C09100=1017.459,-55.888,398.347,165.702,54.848,159.813
C09101=1017.465,-55.638,398.336,165.706,54.842,159.813
C09102=1017.470,-55.388,398.326,165.708,54.836,159.812
C09103=1017.475,-55.139,398.315,165.712,54.830,159.812
C09104=1017.481,-54.889,398.305,165.714,54.824,159.811
C09105=1017.486,-54.640,398.294,165.717,54.817,159.810
C09106=1017.491,-54.389,398.284,165.721,54.811,159.810
C09107=1017.497,-54.140,398.273,165.723,54.805,159.810
C09108=1017.503,-53.863,398.261,165.726,54.798,159.809
C09109=1017.509,-53.585,398.250,165.729,54.791,159.808
C09110=1017.515,-53.308,398.237,165.733,54.784,159.808
C09111=1017.522,-53.030,398.226,165.737,54.777,159.808
C09112=1017.527,-52.780,398.216,165.739,54.771,159.807
C09113=1017.533,-52.531,398.205,165.741,54.765,159.806
C09114=1017.539,-52.281,398.194,165.745,54.759,159.806
C09115=1017.543,-52.032,398.184,165.748,54.752,159.805
C09116=1017.549,-51.782,398.173,165.751,54.746,159.805
C09117=1017.554,-51.532,398.162,165.753,54.739,159.804
C09118=1017.560,-51.282,398.151,165.757,54.733,159.804
C09119=1017.565,-51.033,398.141,165.759,54.727,159.803
C09120=1017.571,-50.783,398.130,165.762,54.721,159.803
C09121=1017.576,-50.533,398.118,165.766,54.715,159.803
C09122=1017.582,-50.283,398.108,165.768,54.709,159.802
C09123=1017.587,-50.034,398.097,165.771,54.703,159.802
C09124=1017.592,-49.784,398.086,165.775,54.697,159.801
C09125=1017.597,-49.534,398.074,165.777,54.691,159.801
C09126=1017.603,-49.285,398.063,165.780,54.685,159.800
C09127=1017.608,-49.035,398.052,165.783,54.678,159.800
C09128=1017.614,-48.785,398.041,165.786,54.673,159.799
C09129=1017.619,-48.536,398.030,165.789,54.667,159.799
C09130=1017.625,-48.286,398.019,165.791,54.661,159.798
C09131=1017.630,-48.036,398.007,165.795,54.655,159.798
C09132=1017.635,-47.787,397.996,165.797,54.649,159.797
C09133=1017.640,-47.536,397.986,165.800,54.643,159.797
C09134=1017.646,-47.287,397.975,165.803,54.636,159.797
C09135=1017.651,-47.037,397.963,165.806,54.631,159.796
C09136=1017.656,-46.788,397.952,165.808,54.624,159.796
C09137=1017.661,-46.538,397.941,165.812,54.618,159.795
C09138=1017.667,-46.288,397.930,165.815,54.612,159.795
C09139=1017.672,-46.039,397.919,165.817,54.606,159.794
C09140=1017.678,-45.789,397.908,165.821,54.600,159.794
C09141=1017.683,-45.539,397.896,165.823,54.594,159.793
C09142=1017.689,-45.289,397.885,165.826,54.588,159.793
C09143=1017.694,-45.039,397.873,165.828,54.582,159.792
C09144=1017.700,-44.790,397.863,165.832,54.576,159.792
C09145=1017.705,-44.540,397.851,165.834,54.570,159.791
C09146=1017.711,-44.291,397.840,165.837,54.563,159.791
C09147=1017.716,-44.041,397.829,165.841,54.557,159.790
C09148=1017.722,-43.792,397.817,165.843,54.551,159.790
C09149=1017.727,-43.542,397.806,165.846,54.546,159.789
C09150=1017.733,-43.293,397.795,165.849,54.539,159.789
C09151=1017.738,-43.043,397.783,165.852,54.533,159.789
C09152=1017.744,-42.793,397.772,165.854,54.527,159.788
C09153=1017.749,-42.543,397.761,165.858,54.520,159.787
C09154=1017.755,-42.293,397.750,165.861,54.515,159.787
C09155=1017.760,-42.043,397.738,165.864,54.508,159.787
C09156=1017.765,-41.794,397.727,165.866,54.502,159.786
C09157=1017.770,-41.544,397.716,165.869,54.496,159.785
C09158=1017.776,-41.295,397.705,165.873,54.490,159.785
C09159=1017.782,-41.045,397.693,165.875,54.483,159.784
C09160=1017.788,-40.795,397.682,165.878,54.478,159.784
C09161=1017.793,-40.546,397.670,165.881,54.471,159.783
C09162=1017.798,-40.296,397.659,165.883,54.465,159.783
C09163=1017.803,-40.046,397.648,165.886,54.459,159.782
C09164=1017.809,-39.797,397.637,165.890,54.453,159.782
C09165=1017.815,-39.547,397.624,165.892,54.446,159.781
C09166=1017.820,-39.297,397.613,165.895,54.441,159.781
C09167=1017.826,-39.048,397.602,165.898,54.434,159.780
C09168=1017.831,-38.798,397.591,165.901,54.429,159.780
C09169=1017.836,-38.549,397.578,165.903,54.422,159.779
C09170=1017.842,-38.298,397.567,165.906,54.417,159.779
C09171=1017.847,-38.048,397.555,165.910,54.410,159.779
C09172=1017.853,-37.772,397.542,165.913,54.404,159.778
C09173=1017.859,-37.495,397.529,165.915,54.397,159.777
C09174=1017.865,-37.217,397.516,165.919,54.391,159.777
C09175=1017.871,-36.940,397.503,165.922,54.384,159.776
C09176=1017.876,-36.690,397.491,165.924,54.378,159.776
C09177=1017.882,-36.441,397.480,165.928,54.371,159.775
C09178=1017.887,-36.191,397.468,165.931,54.366,159.775
C09179=1017.893,-35.942,397.456,165.933,54.359,159.774
C09180=1017.898,-35.691,397.444,165.936,54.354,159.774
C09181=1017.904,-35.442,397.434,165.939,54.347,159.773
C09182=1017.909,-35.193,397.421,165.942,54.342,159.773
C09183=1017.914,-34.943,397.410,165.945,54.335,159.772
C09184=1017.920,-34.693,397.397,165.948,54.329,159.772
C09185=1017.925,-34.443,397.386,165.951,54.323,159.771
C09186=1017.931,-34.194,397.374,165.953,54.317,159.771
C09187=1017.937,-33.944,397.362,165.955,54.311,159.770
C09188=1017.942,-33.695,397.350,165.959,54.305,159.770
C09189=1017.947,-33.445,397.339,165.962,54.298,159.769
C09190=1017.952,-33.196,397.327,165.965,54.293,159.769
C09191=1017.959,-32.945,397.315,165.968,54.286,159.768
C09192=1017.964,-32.696,397.303,165.970,54.280,159.768
C09193=1017.969,-32.446,397.292,165.973,54.274,159.767
C09194=1017.975,-32.197,397.279,165.976,54.268,159.767
C09195=1017.980,-31.947,397.268,165.979,54.262,159.766
C09196=1017.985,-31.698,397.255,165.982,54.256,159.766
C09197=1017.992,-31.447,397.244,165.984,54.250,159.765
C09198=1017.997,-31.198,397.232,165.988,54.243,159.765
C09199=1018.002,-30.948,397.221,165.990,54.238,159.764
C09200=1018.008,-30.698,397.208,165.993,54.231,159.764
C09201=1018.013,-30.449,397.197,165.996,54.225,159.763
C09202=1018.020,-30.199,397.185,165.999,54.219,159.763
C09203=1018.025,-29.949,397.173,166.001,54.213,159.762
C09204=1018.030,-29.700,397.161,166.004,54.207,159.761
C09205=1018.036,-29.450,397.148,166.007,54.200,159.761
C09206=1018.041,-29.200,397.137,166.010,54.195,159.761
C09207=1018.047,-28.951,397.125,166.012,54.188,159.760
C09208=1018.052,-28.701,397.113,166.016,54.182,159.759
C09209=1018.058,-28.452,397.101,166.018,54.176,159.759
C09210=1018.064,-28.202,397.089,166.021,54.169,159.758
C09211=1018.069,-27.952,397.077,166.025,54.163,159.758
C09212=1018.075,-27.702,397.065,166.027,54.157,159.757
C09213=1018.080,-27.452,397.053,166.029,54.151,159.757
C09214=1018.085,-27.203,397.041,166.032,54.145,159.756
C09215=1018.091,-26.953,397.028,166.036,54.139,159.756
C09216=1018.096,-26.704,397.016,166.038,54.133,159.755
C09217=1018.102,-26.454,397.004,166.041,54.127,159.755
C09218=1018.107,-26.205,396.992,166.043,54.121,159.754
C09219=1018.113,-25.955,396.980,166.047,54.115,159.754
C09220=1018.118,-25.706,396.968,166.050,54.109,159.753
C09221=1018.124,-25.456,396.955,166.052,54.103,159.753
C09222=1018.129,-25.206,396.943,166.055,54.097,159.752
C09223=1018.134,-24.956,396.930,166.057,54.091,159.751
C09224=1018.140,-24.706,396.918,166.061,54.085,159.751
C09225=1018.145,-24.457,396.906,166.063,54.079,159.751
C09226=1018.151,-24.207,396.893,166.066,54.072,159.750
C09227=1018.156,-23.958,396.881,166.069,54.067,159.750
C09228=1018.162,-23.708,396.869,166.072,54.060,159.749
C09229=1018.167,-23.459,396.856,166.075,54.055,159.749
C09230=1018.173,-23.209,396.845,166.077,54.049,159.748
C09231=1018.178,-22.959,396.832,166.080,54.042,159.747
C09232=1018.184,-22.710,396.820,166.083,54.036,159.747
C09233=1018.189,-22.460,396.807,166.086,54.030,159.746
C09234=1018.195,-22.210,396.795,166.089,54.024,159.746
C09235=1018.200,-21.961,396.782,166.091,54.018,159.745
C09236=1018.206,-21.683,396.769,166.094,54.011,159.745
C09237=1018.213,-21.405,396.754,166.098,54.005,159.744
C09238=1018.219,-21.127,396.741,166.101,53.997,159.743
C09239=1018.225,-20.848,396.727,166.104,53.991,159.743
C09240=1018.230,-20.598,396.714,166.107,53.984,159.742
C09241=1018.236,-20.349,396.702,166.109,53.978,159.742
C09242=1018.242,-20.099,396.690,166.112,53.973,159.741
C09243=1018.247,-19.850,396.678,166.115,53.966,159.741
C09244=1018.253,-19.600,396.665,166.118,53.960,159.740
C09245=1018.258,-19.351,396.653,166.120,53.954,159.740
C09246=1018.264,-19.101,396.640,166.123,53.948,159.739
C09247=1018.269,-18.851,396.627,166.126,53.942,159.739
C09248=1018.275,-18.602,396.615,166.129,53.935,159.738
C09249=1018.280,-18.352,396.602,166.131,53.929,159.737
C09250=1018.286,-18.103,396.590,166.134,53.924,159.737
C09251=1018.292,-17.853,396.578,166.138,53.917,159.736
C09252=1018.298,-17.603,396.565,166.140,53.911,159.736
C09253=1018.303,-17.354,396.553,166.142,53.905,159.735
C09254=1018.309,-17.104,396.540,166.146,53.898,159.735
C09255=1018.314,-16.855,396.528,166.149,53.893,159.734
C09256=1018.319,-16.605,396.515,166.151,53.886,159.734
C09257=1018.325,-16.355,396.502,166.154,53.880,159.733
C09258=1018.331,-16.106,396.490,166.157,53.874,159.732
C09259=1018.336,-15.856,396.478,166.159,53.867,159.732
C09260=1018.343,-15.606,396.464,166.162,53.862,159.731
C09261=1018.347,-15.357,396.452,166.165,53.856,159.731
C09262=1018.353,-15.107,396.439,166.167,53.850,159.730
C09263=1018.358,-14.857,396.426,166.171,53.844,159.730
C09264=1018.364,-14.608,396.413,166.174,53.837,159.729
C09265=1018.370,-14.358,396.400,166.176,53.831,159.729
C09266=1018.374,-14.109,396.388,166.179,53.826,159.728
C09267=1018.380,-13.859,396.375,166.181,53.820,159.728
C09268=1018.388,-13.518,396.357,166.185,53.811,159.727
C09269=1018.396,-13.177,396.340,166.188,53.803,159.726
C09270=1018.403,-12.835,396.322,166.194,53.795,159.725
C09271=1018.410,-12.493,396.304,166.197,53.786,159.725
C09272=1018.416,-12.245,396.291,166.200,53.780,159.724
C09273=1018.421,-11.995,396.278,166.202,53.774,159.723
C09274=1018.427,-11.745,396.266,166.205,53.769,159.723
C09275=1018.433,-11.496,396.253,166.207,53.762,159.722
C09276=1018.438,-11.246,396.240,166.211,53.756,159.722
C09277=1018.444,-10.996,396.227,166.213,53.750,159.721
C09278=1018.449,-10.747,396.214,166.216,53.743,159.721
C09279=1018.455,-10.497,396.201,166.218,53.738,159.720
C09280=1018.460,-10.247,396.189,166.221,53.732,159.719
C09281=1018.466,-9.998,396.175,166.224,53.725,159.719
C09282=1018.471,-9.749,396.163,166.227,53.719,159.718
C09283=1018.476,-9.499,396.149,166.230,53.714,159.718
C09284=1018.483,-9.249,396.136,166.232,53.707,159.717
C09285=1018.489,-8.999,396.124,166.235,53.701,159.717
C09286=1018.493,-8.751,396.110,166.238,53.695,159.716
C09287=1018.499,-8.501,396.097,166.241,53.688,159.716
C09288=1018.505,-8.250,396.084,166.243,53.683,159.715
C09289=1018.511,-8.001,396.071,166.246,53.677,159.714
C09290=1018.517,-7.751,396.059,166.248,53.671,159.714
C09291=1018.522,-7.502,396.045,166.252,53.664,159.713
C09292=1018.527,-7.253,396.032,166.254,53.658,159.713
C09293=1018.533,-7.003,396.019,166.257,53.652,159.712
C09294=1018.539,-6.753,396.006,166.259,53.646,159.711
C09295=1018.544,-6.503,395.993,166.263,53.640,159.711
C09296=1018.549,-6.285,395.982,166.264,53.634,159.710
C09297=1018.554,-6.066,395.970,166.267,53.628,159.710
C09298=1018.559,-5.847,395.959,166.269,53.623,159.709
C09299=1018.563,-5.628,395.947,166.272,53.618,159.709
C09300=1018.569,-5.409,395.936,166.275,53.612,159.709
C09301=1018.574,-5.191,395.924,166.277,53.607,159.708
C09302=1018.578,-4.971,395.913,166.279,53.601,159.707
C09303=1018.583,-4.752,395.902,166.281,53.596,159.707
C09304=1018.590,-4.503,395.888,166.285,53.590,159.706
C09305=1018.595,-4.253,395.875,166.287,53.583,159.706
C09306=1018.600,-4.003,395.861,166.290,53.578,159.705
C09307=1018.606,-3.754,395.848,166.293,53.572,159.705
C09308=1018.612,-3.504,395.835,166.295,53.566,159.704
C09309=1018.617,-3.254,395.821,166.298,53.560,159.703
C09310=1018.622,-3.005,395.807,166.300,53.554,159.703
C09311=1018.628,-2.755,395.795,166.303,53.548,159.702
C09312=1018.633,-2.506,395.781,166.306,53.542,159.702
C09313=1018.639,-2.256,395.767,166.308,53.536,159.701
C09314=1018.644,-2.007,395.753,166.312,53.530,159.701
C09315=1018.649,-1.757,395.740,166.315,53.524,159.700
C09316=1018.656,-1.507,395.727,166.317,53.518,159.700
C09317=1018.660,-1.258,395.713,166.319,53.512,159.699
C09318=1018.666,-1.009,395.700,166.322,53.506,159.698
C09319=1018.671,-0.759,395.686,166.325,53.500,159.698
C09320=1018.677,-0.509,395.673,166.327,53.494,159.697
C09321=1018.683,-0.260,395.659,166.330,53.488,159.697
C09322=1018.688,-0.010,395.645,166.333,53.483,159.696
C09323=1018.694,0.239,395.632,166.336,53.476,159.696
C09324=1018.699,0.490,395.618,166.339,53.470,159.695
C09325=1018.705,0.739,395.605,166.341,53.464,159.694
C09326=1018.711,0.988,395.591,166.344,53.458,159.694
C09327=1018.716,1.238,395.577,166.347,53.452,159.693
C09328=1018.721,1.487,395.564,166.349,53.446,159.693
C09329=1018.726,1.737,395.551,166.351,53.440,159.692
C09330=1018.732,1.986,395.537,166.354,53.434,159.691
C09331=1018.738,2.236,395.524,166.358,53.428,159.691
C09332=1018.743,2.485,395.510,166.360,53.422,159.690
C09333=1018.749,2.735,395.496,166.363,53.416,159.690
C09334=1018.754,2.985,395.482,166.365,53.409,159.689
C09335=1018.760,3.234,395.469,166.368,53.403,159.688
C09336=1018.766,3.484,395.456,166.370,53.397,159.688
C09337=1018.771,3.734,395.442,166.373,53.392,159.687
C09338=1018.777,3.983,395.428,166.376,53.386,159.687
C09339=1018.782,4.233,395.414,166.379,53.379,159.686
C09340=1018.788,4.482,395.401,166.382,53.373,159.686
C09341=1018.794,4.732,395.387,166.384,53.367,159.685
C09342=1018.799,4.981,395.373,166.387,53.361,159.684
C09343=1018.805,5.231,395.359,166.389,53.354,159.684
C09344=1018.810,5.480,395.345,166.392,53.348,159.683
C09345=1018.816,5.730,395.332,166.395,53.343,159.683
C09346=1018.822,5.980,395.319,166.398,53.336,159.682
C09347=1018.827,6.229,395.305,166.401,53.330,159.681
C09348=1018.833,6.479,395.291,166.403,53.324,159.681
C09349=1018.838,6.729,395.277,166.405,53.318,159.680
C09350=1018.844,6.978,395.264,166.408,53.312,159.680
C09351=1018.850,7.227,395.250,166.410,53.306,159.679
C09352=1018.855,7.477,395.236,166.414,53.299,159.678
C09353=1018.861,7.727,395.222,166.416,53.293,159.678
C09354=1018.866,7.976,395.209,166.419,53.287,159.677
C09355=1018.872,8.225,395.195,166.421,53.281,159.676
C09356=1018.878,8.475,395.181,166.424,53.275,159.676
C09357=1018.883,8.724,395.168,166.426,53.269,159.675
C09358=1018.889,8.975,395.153,166.430,53.262,159.675
C09359=1018.895,9.224,395.139,166.433,53.257,159.674
C09360=1018.901,9.474,395.126,166.435,53.250,159.674
C09361=1018.907,9.723,395.112,166.438,53.244,159.673
C09362=1018.912,9.973,395.098,166.440,53.238,159.672
C09363=1018.917,10.222,395.085,166.443,53.232,159.672
C09364=1018.924,10.503,395.069,166.446,53.225,159.671
C09365=1018.930,10.785,395.053,166.449,53.218,159.670
C09366=1018.937,11.067,395.038,166.452,53.210,159.669
C09367=1018.944,11.349,395.022,166.455,53.203,159.669
C09368=1018.949,11.599,395.008,166.458,53.197,159.668
C09369=1018.955,11.849,394.994,166.460,53.191,159.667
C09370=1018.961,12.098,394.981,166.463,53.185,159.667
C09371=1018.966,12.347,394.967,166.466,53.178,159.666
C09372=1018.972,12.597,394.953,166.469,53.172,159.666
C09373=1018.977,12.847,394.939,166.471,53.166,159.665
C09374=1018.983,13.096,394.925,166.474,53.160,159.664
C09375=1018.989,13.346,394.910,166.476,53.154,159.664
C09376=1018.995,13.595,394.896,166.479,53.148,159.663
C09377=1019.000,13.845,394.882,166.482,53.141,159.663
C09378=1019.006,14.094,394.869,166.485,53.135,159.662
C09379=1019.011,14.343,394.854,166.488,53.130,159.661
C09380=1019.017,14.593,394.840,166.490,53.124,159.661
C09381=1019.022,14.843,394.826,166.493,53.118,159.660
C09382=1019.029,15.092,394.811,166.495,53.111,159.659
C09383=1019.034,15.342,394.797,166.498,53.105,159.659
C09384=1019.039,15.592,394.783,166.500,53.099,159.658
C09385=1019.044,15.841,394.769,166.503,53.093,159.658
C09386=1019.050,16.090,394.755,166.505,53.087,159.657
C09387=1019.056,16.340,394.741,166.509,53.081,159.656
C09388=1019.062,16.590,394.726,166.511,53.074,159.656
C09389=1019.067,16.839,394.712,166.514,53.068,159.655
C09390=1019.073,17.089,394.698,166.516,53.062,159.654
C09391=1019.079,17.338,394.683,166.519,53.056,159.654
C09392=1019.084,17.587,394.670,166.521,53.050,159.653
C09393=1019.090,17.838,394.655,166.524,53.045,159.653
C09394=1019.095,18.087,394.640,166.527,53.039,159.652
C09395=1019.101,18.336,394.626,166.529,53.032,159.651
C09396=1019.106,18.586,394.612,166.533,53.026,159.651
C09397=1019.113,18.835,394.597,166.536,53.020,159.650
C09398=1019.118,19.085,394.584,166.538,53.014,159.650
C09399=1019.124,19.334,394.569,166.541,53.008,159.649
C09400=1019.129,19.584,394.555,166.543,53.002,159.648
C09401=1019.134,19.833,394.540,166.546,52.995,159.648
C09402=1019.141,20.083,394.526,166.548,52.989,159.647
C09403=1019.146,20.332,394.511,166.551,52.983,159.646
C09404=1019.151,20.582,394.497,166.553,52.977,159.646
C09405=1019.157,20.831,394.482,166.556,52.971,159.645
C09406=1019.163,21.081,394.468,166.558,52.965,159.644
C09407=1019.168,21.330,394.453,166.561,52.959,159.644
C09408=1019.173,21.580,394.439,166.564,52.952,159.643
C09409=1019.179,21.829,394.424,166.567,52.946,159.643
C09410=1019.185,22.079,394.410,166.569,52.940,159.642
C09411=1019.190,22.329,394.395,166.572,52.934,159.641
C09412=1019.196,22.578,394.381,166.574,52.928,159.641
C09413=1019.202,22.828,394.366,166.577,52.922,159.640
C09414=1019.208,23.077,394.352,166.580,52.916,159.639
C09415=1019.213,23.327,394.337,166.582,52.910,159.639
C09416=1019.219,23.576,394.322,166.585,52.904,159.638
C09417=1019.225,23.826,394.308,166.587,52.898,159.637
C09418=1019.230,24.075,394.294,166.590,52.892,159.637
C09419=1019.235,24.325,394.279,166.593,52.885,159.636
C09420=1019.241,24.574,394.264,166.596,52.879,159.636
C09421=1019.247,24.823,394.250,166.598,52.873,159.635
C09422=1019.252,25.073,394.235,166.601,52.867,159.634
C09423=1019.258,25.323,394.220,166.603,52.861,159.634
C09424=1019.264,25.572,394.206,166.606,52.855,159.633
C09425=1019.270,25.821,394.192,166.608,52.849,159.632
C09426=1019.275,26.071,394.176,166.611,52.843,159.632
C09427=1019.281,26.321,394.162,166.614,52.836,159.631
C09428=1019.287,26.605,394.145,166.617,52.829,159.630
C09429=1019.294,26.887,394.129,166.620,52.822,159.630
C09430=1019.300,27.171,394.112,166.623,52.816,159.629
C09431=1019.306,27.454,394.095,166.626,52.809,159.628
C09432=1019.312,27.703,394.080,166.629,52.803,159.628
C09433=1019.317,27.953,394.066,166.632,52.796,159.627
C09434=1019.323,28.203,394.051,166.634,52.790,159.626
C09435=1019.329,28.452,394.036,166.637,52.784,159.626
C09436=1019.334,28.701,394.021,166.639,52.778,159.625
C09437=1019.340,28.951,394.006,166.642,52.772,159.624
C09438=1019.345,29.201,393.992,166.644,52.766,159.624
C09439=1019.351,29.451,393.976,166.647,52.760,159.623
C09440=1019.357,29.700,393.962,166.650,52.754,159.623
C09441=1019.362,29.949,393.946,166.652,52.748,159.622
C09442=1019.368,30.199,393.931,166.655,52.742,159.621
C09443=1019.373,30.448,393.916,166.657,52.736,159.621
C09444=1019.379,30.698,393.902,166.660,52.730,159.620
C09445=1019.384,30.947,393.887,166.662,52.724,159.619
C09446=1019.390,31.196,393.872,166.665,52.718,159.619
C09447=1019.396,31.446,393.857,166.667,52.712,159.618
C09448=1019.402,31.695,393.842,166.670,52.705,159.617
C09449=1019.407,31.945,393.827,166.673,52.699,159.617
C09450=1019.412,32.194,393.811,166.675,52.693,159.616
C09451=1019.418,32.443,393.797,166.679,52.687,159.616
C09452=1019.423,32.694,393.782,166.681,52.681,159.615
C09453=1019.429,32.943,393.767,166.684,52.675,159.614
C09454=1019.435,33.193,393.752,166.686,52.669,159.614
C09455=1019.441,33.442,393.737,166.689,52.663,159.613
C09456=1019.446,33.692,393.722,166.692,52.657,159.612
C09457=1019.452,33.941,393.707,166.694,52.651,159.612
C09458=1019.458,34.191,393.692,166.696,52.644,159.611
C09459=1019.464,34.440,393.677,166.699,52.638,159.610
C09460=1019.469,34.690,393.662,166.701,52.632,159.609
C09461=1019.475,34.939,393.647,166.704,52.626,159.609
C09462=1019.480,35.188,393.632,166.707,52.620,159.608
C09463=1019.486,35.438,393.617,166.709,52.614,159.608
C09464=1019.491,35.687,393.602,166.713,52.607,159.607
C09465=1019.498,35.936,393.587,166.715,52.601,159.606
C09466=1019.503,36.186,393.572,166.718,52.595,159.606
C09467=1019.508,36.436,393.556,166.720,52.588,159.605
C09468=1019.514,36.685,393.541,166.723,52.582,159.604
C09469=1019.520,36.935,393.526,166.725,52.576,159.604
C09470=1019.526,37.185,393.510,166.728,52.570,159.603
C09471=1019.531,37.434,393.495,166.730,52.564,159.602
C09472=1019.537,37.684,393.480,166.733,52.558,159.602
C09473=1019.542,37.933,393.465,166.735,52.552,159.601
C09474=1019.548,38.183,393.450,166.738,52.546,159.600
C09475=1019.553,38.431,393.434,166.741,52.540,159.600
C09476=1019.559,38.681,393.419,166.743,52.534,159.599
C09477=1019.564,38.930,393.404,166.746,52.528,159.598
C09478=1019.570,39.180,393.388,166.748,52.522,159.598
C09479=1019.575,39.430,393.373,166.751,52.516,159.597
C09480=1019.581,39.680,393.357,166.754,52.510,159.596
C09481=1019.587,39.928,393.342,166.756,52.504,159.596
C09482=1019.593,40.178,393.326,166.759,52.498,159.595
C09483=1019.598,40.427,393.311,166.761,52.492,159.594
C09484=1019.603,40.677,393.296,166.764,52.486,159.594
C09485=1019.608,40.926,393.281,166.766,52.480,159.593
C09486=1019.615,41.175,393.265,166.769,52.474,159.592
C09487=1019.621,41.425,393.249,166.773,52.467,159.592
C09488=1019.626,41.675,393.234,166.775,52.461,159.591
C09489=1019.631,41.925,393.219,166.777,52.454,159.590
C09490=1019.637,42.173,393.203,166.780,52.448,159.590
C09491=1019.643,42.423,393.188,166.783,52.442,159.589
C09492=1019.649,42.706,393.170,166.785,52.436,159.588
C09493=1019.656,42.990,393.152,166.788,52.429,159.588
C09494=1019.661,43.273,393.134,166.792,52.422,159.587
C09495=1019.668,43.555,393.116,166.794,52.415,159.586
C09496=1019.673,43.805,393.101,166.796,52.409,159.585
C09497=1019.679,44.055,393.085,166.799,52.403,159.585
C09498=1019.684,44.304,393.069,166.802,52.397,159.584
C09499=1019.690,44.554,393.054,166.804,52.391,159.584
C09500=1019.695,44.803,393.038,166.807,52.385,159.583
C09501=1019.700,45.053,393.022,166.809,52.379,159.582
C09502=1019.706,45.302,393.006,166.812,52.373,159.582
C09503=1019.711,45.552,392.990,166.815,52.367,159.581
C09504=1019.717,45.802,392.975,166.817,52.361,159.580
C09505=1019.722,46.050,392.959,166.820,52.355,159.580
C09506=1019.728,46.300,392.943,166.822,52.349,159.579
C09507=1019.734,46.550,392.927,166.825,52.343,159.578
C09508=1019.739,46.799,392.912,166.828,52.337,159.578
C09509=1019.745,47.048,392.896,166.830,52.331,159.577
C09510=1019.750,47.298,392.880,166.833,52.325,159.576
C09511=1019.756,47.547,392.864,166.835,52.319,159.576
C09512=1019.761,47.797,392.849,166.838,52.313,159.575
C09513=1019.767,48.045,392.833,166.841,52.307,159.574
C09514=1019.772,48.296,392.817,166.843,52.301,159.574
C09515=1019.777,48.545,392.800,166.846,52.295,159.573
C09516=1019.783,48.794,392.785,166.848,52.289,159.572
C09517=1019.788,49.044,392.769,166.851,52.283,159.572
C09518=1019.794,49.294,392.753,166.854,52.277,159.571
C09519=1019.799,49.542,392.738,166.856,52.270,159.570
C09520=1019.805,49.792,392.722,166.859,52.264,159.570
C09521=1019.811,50.042,392.706,166.861,52.258,159.569
C09522=1019.817,50.291,392.690,166.864,52.252,159.568
C09523=1019.822,50.540,392.674,166.866,52.246,159.568
C09524=1019.828,50.789,392.658,166.869,52.240,159.567
C09525=1019.833,51.040,392.642,166.872,52.234,159.566
C09526=1019.838,51.288,392.626,166.875,52.227,159.566
C09527=1019.844,51.538,392.610,166.877,52.221,159.565
C09528=1019.850,51.788,392.594,166.880,52.215,159.564
C09529=1019.855,52.036,392.578,166.883,52.209,159.564
C09530=1019.861,52.286,392.563,166.885,52.203,159.563
C09531=1019.867,52.536,392.547,166.888,52.197,159.562
C09532=1019.873,52.785,392.530,166.890,52.190,159.562
C09533=1019.878,53.034,392.515,166.893,52.184,159.561
C09534=1019.884,53.284,392.499,166.895,52.178,159.560
C09535=1019.889,53.534,392.483,166.898,52.172,159.560
C09536=1019.895,53.783,392.467,166.901,52.166,159.559
C09537=1019.900,54.032,392.451,166.903,52.160,159.558
C09538=1019.906,54.282,392.435,166.905,52.154,159.557
C09539=1019.912,54.531,392.419,166.908,52.148,159.557
C09540=1019.918,54.781,392.403,166.911,52.142,159.556
C09541=1019.923,55.030,392.387,166.914,52.135,159.555
C09542=1019.929,55.279,392.371,166.917,52.129,159.555
C09543=1019.934,55.529,392.355,166.919,52.123,159.554
C09544=1019.940,55.779,392.339,166.922,52.117,159.553
C09545=1019.946,56.028,392.323,166.924,52.110,159.553
C09546=1019.951,56.277,392.307,166.927,52.104,159.552
C09547=1019.957,56.526,392.290,166.929,52.098,159.551
C09548=1019.962,56.776,392.275,166.932,52.092,159.551
C09549=1019.968,57.026,392.259,166.934,52.085,159.550
C09550=1019.974,57.275,392.242,166.937,52.079,159.549
C09551=1019.979,57.524,392.227,166.941,52.073,159.549
C09552=1019.985,57.773,392.211,166.943,52.066,159.548
C09553=1019.991,58.023,392.195,166.945,52.060,159.547
C09554=1019.997,58.272,392.178,166.948,52.054,159.546
C09555=1020.002,58.522,392.162,166.950,52.048,159.545
C09556=1020.009,58.805,392.144,166.954,52.041,159.545
C09557=1020.016,59.088,392.126,166.957,52.034,159.544
C09558=1020.022,59.371,392.107,166.959,52.027,159.543
C09559=1020.028,59.654,392.090,166.962,52.020,159.542
C09560=1020.034,59.904,392.073,166.965,52.013,159.542
C09561=1020.040,60.153,392.056,166.968,52.007,159.541
C09562=1020.045,60.403,392.041,166.970,52.000,159.540
C09563=1020.051,60.653,392.025,166.973,51.994,159.540
C09564=1020.057,60.901,392.009,166.976,51.988,159.539
C09565=1020.062,61.150,391.992,166.978,51.982,159.538
C09566=1020.068,61.400,391.976,166.981,51.976,159.537
C09567=1020.074,61.649,391.960,166.983,51.970,159.537
C09568=1020.080,61.899,391.944,166.987,51.963,159.536
C09569=1020.085,62.149,391.928,166.989,51.957,159.535
C09570=1020.091,62.398,391.911,166.991,51.950,159.534
C09571=1020.097,62.648,391.895,166.994,51.944,159.534
C09572=1020.103,62.897,391.879,166.996,51.937,159.533
C09573=1020.108,63.146,391.863,166.999,51.931,159.532
C09574=1020.114,63.395,391.846,167.002,51.926,159.532
C09575=1020.120,63.645,391.830,167.004,51.920,159.531
C09576=1020.125,63.894,391.813,167.007,51.913,159.530
C09577=1020.131,64.144,391.797,167.010,51.907,159.530
C09578=1020.136,64.393,391.780,167.013,51.901,159.529
C09579=1020.142,64.643,391.764,167.016,51.895,159.528
C09580=1020.148,64.892,391.747,167.018,51.888,159.527
C09581=1020.153,65.142,391.730,167.020,51.882,159.527
C09582=1020.159,65.391,391.714,167.023,51.876,159.526
C09583=1020.164,65.641,391.697,167.025,51.869,159.525
C09584=1020.170,65.890,391.681,167.028,51.863,159.525
C09585=1020.175,66.139,391.665,167.031,51.858,159.524
C09586=1020.181,66.388,391.648,167.033,51.852,159.523
C09587=1020.186,66.638,391.632,167.036,51.845,159.522
C09588=1020.192,66.887,391.615,167.038,51.839,159.522
C09589=1020.198,67.136,391.598,167.041,51.833,159.521
C09590=1020.203,67.386,391.581,167.043,51.826,159.520
C09591=1020.209,67.635,391.565,167.047,51.820,159.520
C09592=1020.215,67.885,391.548,167.050,51.814,159.519
C09593=1020.221,68.134,391.532,167.052,51.808,159.518
C09594=1020.226,68.384,391.515,167.055,51.801,159.518
C09595=1020.231,68.633,391.498,167.057,51.796,159.517
C09596=1020.237,68.882,391.481,167.060,51.790,159.516
C09597=1020.242,69.132,391.465,167.063,51.784,159.516
C09598=1020.248,69.381,391.448,167.065,51.777,159.515
C09599=1020.254,69.631,391.431,167.068,51.771,159.514
C09600=1020.259,69.880,391.414,167.070,51.765,159.513
C09601=1020.265,70.129,391.398,167.072,51.758,159.513
C09602=1020.270,70.379,391.381,167.075,51.753,159.512
C09603=1020.276,70.628,391.365,167.078,51.747,159.511
C09604=1020.282,70.877,391.347,167.081,51.741,159.511
C09605=1020.287,71.127,391.330,167.083,51.734,159.510
C09606=1020.293,71.376,391.314,167.085,51.728,159.509
C09607=1020.298,71.626,391.297,167.089,51.722,159.509
C09608=1020.304,71.875,391.279,167.092,51.716,159.508
C09609=1020.310,72.124,391.263,167.094,51.709,159.507
C09610=1020.315,72.374,391.246,167.097,51.703,159.506
C09611=1020.320,72.623,391.229,167.100,51.697,159.506
C09612=1020.326,72.872,391.212,167.102,51.691,159.505
C09613=1020.331,73.122,391.196,167.104,51.685,159.504
C09614=1020.337,73.371,391.178,167.107,51.679,159.504
C09615=1020.343,73.620,391.162,167.109,51.672,159.503
C09616=1020.348,73.870,391.145,167.112,51.666,159.502
C09617=1020.354,74.119,391.127,167.115,51.660,159.501
C09618=1020.360,74.368,391.111,167.117,51.654,159.500
C09619=1020.365,74.617,391.094,167.121,51.647,159.500
C09620=1020.371,74.900,391.075,167.123,51.641,159.499
C09621=1020.378,75.184,391.055,167.126,51.634,159.498
C09622=1020.384,75.467,391.036,167.129,51.626,159.497
C09623=1020.391,75.749,391.017,167.133,51.619,159.497
C09624=1020.396,75.999,391.000,167.135,51.613,159.496
C09625=1020.402,76.249,390.983,167.138,51.607,159.495
C09626=1020.407,76.499,390.966,167.140,51.601,159.494
C09627=1020.413,76.748,390.948,167.143,51.595,159.494
C09628=1020.419,76.997,390.932,167.146,51.589,159.493
C09629=1020.424,77.246,390.914,167.148,51.582,159.492
C09630=1020.429,77.496,390.897,167.151,51.576,159.492
C09631=1020.435,77.745,390.880,167.153,51.570,159.491
C09632=1020.440,77.994,390.863,167.156,51.564,159.490
C09633=1020.446,78.243,390.845,167.158,51.558,159.489
C09634=1020.451,78.492,390.828,167.161,51.552,159.489
C09635=1020.456,78.742,390.811,167.164,51.546,159.488
C09636=1020.462,78.991,390.793,167.166,51.539,159.487
C09637=1020.468,79.241,390.776,167.170,51.533,159.487
C09638=1020.473,79.491,390.759,167.173,51.527,159.486
C09639=1020.479,79.739,390.742,167.175,51.521,159.485
C09640=1020.485,79.989,390.725,167.178,51.515,159.485
C09641=1020.490,80.238,390.707,167.180,51.509,159.484
C09642=1020.495,80.488,390.690,167.183,51.503,159.483
C09643=1020.501,80.737,390.673,167.186,51.497,159.483
C09644=1020.506,80.986,390.655,167.188,51.490,159.482
C09645=1020.512,81.236,390.638,167.191,51.484,159.481
C09646=1020.518,81.485,390.621,167.194,51.479,159.480
C09647=1020.523,81.734,390.603,167.196,51.472,159.480
C09648=1020.528,81.984,390.586,167.199,51.466,159.479
C09649=1020.534,82.233,390.569,167.201,51.460,159.478
C09650=1020.540,82.482,390.551,167.204,51.454,159.477
C09651=1020.545,82.732,390.534,167.206,51.448,159.477
C09652=1020.551,82.981,390.516,167.210,51.441,159.476
C09653=1020.556,83.230,390.499,167.212,51.435,159.475
C09654=1020.562,83.479,390.481,167.215,51.429,159.475
C09655=1020.567,83.729,390.464,167.218,51.423,159.474
C09656=1020.573,83.978,390.447,167.220,51.416,159.473
C09657=1020.578,84.227,390.429,167.223,51.410,159.473
C09658=1020.584,84.477,390.412,167.225,51.404,159.472
C09659=1020.589,84.726,390.394,167.228,51.398,159.471
C09660=1020.595,84.976,390.377,167.231,51.392,159.470
C09661=1020.601,85.225,390.359,167.233,51.386,159.470
C09662=1020.606,85.474,390.342,167.237,51.379,159.469
C09663=1020.612,85.724,390.324,167.239,51.373,159.468
C09664=1020.617,85.973,390.307,167.242,51.367,159.467
C09665=1020.623,86.222,390.289,167.244,51.361,159.467
C09666=1020.628,86.472,390.272,167.247,51.354,159.466
C09667=1020.634,86.720,390.255,167.250,51.348,159.465
C09668=1020.640,86.970,390.237,167.252,51.342,159.464
C09669=1020.646,87.219,390.220,167.255,51.336,159.464
C09670=1020.652,87.468,390.202,167.258,51.330,159.463
C09671=1020.657,87.718,390.186,167.261,51.323,159.462
C09672=1020.663,87.968,390.168,167.263,51.317,159.462
C09673=1020.668,88.217,390.150,167.266,51.311,159.461
C09674=1020.674,88.466,390.132,167.269,51.305,159.460
C09675=1020.679,88.715,390.115,167.271,51.298,159.459
C09676=1020.686,88.965,390.097,167.275,51.292,159.459
C09677=1020.691,89.214,390.080,167.277,51.286,159.458
C09678=1020.696,89.464,390.062,167.280,51.279,159.457
C09679=1020.702,89.713,390.044,167.282,51.274,159.457
C09680=1020.707,89.962,390.026,167.285,51.268,159.456
C09681=1020.712,90.212,390.008,167.288,51.261,159.455
C09682=1020.717,90.461,389.991,167.290,51.255,159.454
C09683=1020.724,90.710,389.973,167.293,51.249,159.454
C09684=1020.729,90.993,389.952,167.296,51.242,159.453
C09685=1020.736,91.276,389.932,167.299,51.235,159.452
C09686=1020.742,91.559,389.912,167.302,51.228,159.451
C09687=1020.749,91.842,389.891,167.305,51.221,159.451
C09688=1020.753,92.091,389.873,167.308,51.216,159.450
C09689=1020.760,92.341,389.855,167.310,51.209,159.449
C09690=1020.765,92.590,389.838,167.313,51.203,159.448
C09691=1020.770,92.839,389.820,167.316,51.197,159.448
C09692=1020.776,93.089,389.802,167.319,51.190,159.447
C09693=1020.781,93.338,389.784,167.322,51.184,159.446
C09694=1020.787,93.587,389.767,167.325,51.179,159.446
C09695=1020.792,93.836,389.748,167.327,51.172,159.445
C09696=1020.798,94.086,389.731,167.330,51.166,159.444
C09697=1020.803,94.335,389.713,167.332,51.160,159.443
C09698=1020.808,94.585,389.695,167.335,51.154,159.443
C09699=1020.815,94.834,389.676,167.338,51.148,159.442
C09700=1020.820,95.083,389.659,167.340,51.141,159.441
C09701=1020.826,95.332,389.641,167.344,51.135,159.441
C09702=1020.831,95.582,389.622,167.346,51.129,159.440
C09703=1020.837,95.831,389.605,167.349,51.123,159.439
C09704=1020.842,96.080,389.587,167.352,51.117,159.438
C09705=1020.847,96.330,389.569,167.354,51.111,159.438
C09706=1020.853,96.578,389.551,167.357,51.104,159.437
C09707=1020.859,96.828,389.533,167.359,51.099,159.436
C09708=1020.865,97.077,389.515,167.363,51.092,159.435
C09709=1020.870,97.326,389.497,167.366,51.086,159.435
C09710=1020.876,97.576,389.479,167.368,51.079,159.434
C09711=1020.881,97.825,389.461,167.371,51.073,159.433
C09712=1020.886,98.074,389.442,167.374,51.068,159.433
C09713=1020.893,98.324,389.425,167.376,51.061,159.432
C09714=1020.898,98.573,389.407,167.380,51.055,159.431
C09715=1020.903,98.823,389.388,167.382,51.048,159.430
C09716=1020.909,99.072,389.371,167.385,51.042,159.430
C09717=1020.915,99.320,389.353,167.387,51.036,159.429
C09718=1020.920,99.570,389.334,167.390,51.030,159.428
C09719=1020.926,99.819,389.317,167.393,51.024,159.428
C09720=1020.931,100.069,389.297,167.395,51.018,159.427
C09721=1020.936,100.318,389.279,167.398,51.012,159.426
C09722=1020.942,100.568,389.261,167.401,51.006,159.425
C09723=1020.947,100.817,389.242,167.404,50.999,159.425
C09724=1020.953,101.066,389.225,167.407,50.993,159.424
C09725=1020.959,101.315,389.205,167.410,50.987,159.423
C09726=1020.963,101.564,389.187,167.412,50.982,159.423
C09727=1020.969,101.814,389.169,167.415,50.975,159.422
C09728=1020.975,102.063,389.151,167.418,50.969,159.421
C09729=1020.980,102.312,389.133,167.420,50.963,159.420
C09730=1020.986,102.561,389.114,167.423,50.957,159.420
C09731=1020.991,102.810,389.096,167.426,50.951,159.419
C09732=1020.997,103.060,389.078,167.429,50.944,159.418
C09733=1021.002,103.309,389.059,167.432,50.938,159.418
C09734=1021.008,103.559,389.041,167.435,50.932,159.417
C09735=1021.013,103.808,389.022,167.437,50.926,159.416
C09736=1021.019,104.057,389.004,167.440,50.920,159.415
C09737=1021.024,104.306,388.985,167.443,50.914,159.415
C09738=1021.029,104.555,388.967,167.445,50.908,159.414
C09739=1021.035,104.805,388.948,167.449,50.901,159.413
C09740=1021.040,105.054,388.930,167.452,50.896,159.413
C09741=1021.047,105.303,388.912,167.454,50.889,159.412
C09742=1021.051,105.552,388.893,167.457,50.883,159.411
C09743=1021.057,105.802,388.874,167.459,50.877,159.410
C09744=1021.063,106.051,388.857,167.462,50.871,159.410
C09745=1021.068,106.300,388.837,167.465,50.865,159.409
C09746=1021.074,106.549,388.820,167.468,50.858,159.408
C09747=1021.079,106.799,388.800,167.471,50.852,159.408
C09748=1021.086,107.082,388.780,167.474,50.845,159.407
C09749=1021.091,107.366,388.759,167.477,50.838,159.406
C09750=1021.098,107.648,388.737,167.480,50.832,159.405
C09751=1021.105,107.932,388.717,167.483,50.825,159.404
C09752=1021.110,108.181,388.697,167.487,50.818,159.404
C09753=1021.116,108.430,388.680,167.490,50.812,159.403
C09754=1021.121,108.679,388.661,167.492,50.806,159.402
C09755=1021.127,108.928,388.643,167.495,50.800,159.401
C09756=1021.133,109.178,388.624,167.497,50.793,159.400
C09757=1021.138,109.427,388.605,167.501,50.787,159.400
C09758=1021.144,109.676,388.587,167.504,50.781,159.399
C09759=1021.149,109.925,388.568,167.506,50.775,159.398
C09760=1021.155,110.175,388.549,167.509,50.769,159.398
C09761=1021.159,110.424,388.531,167.511,50.762,159.397
C09762=1021.165,110.673,388.511,167.514,50.757,159.396
C09763=1021.172,110.922,388.493,167.517,50.751,159.396
C09764=1021.176,111.172,388.475,167.520,50.744,159.395
C09765=1021.182,111.421,388.455,167.523,50.738,159.394
C09766=1021.187,111.670,388.436,167.526,50.732,159.394
C09767=1021.194,111.919,388.418,167.529,50.726,159.393
C09768=1021.198,112.168,388.400,167.531,50.720,159.392
C09769=1021.204,112.418,388.380,167.535,50.713,159.391
C09770=1021.210,112.667,388.361,167.538,50.707,159.391
C09771=1021.215,112.916,388.342,167.540,50.702,159.390
C09772=1021.220,113.165,388.323,167.543,50.696,159.389
C09773=1021.226,113.414,388.304,167.546,50.690,159.389
C09774=1021.231,113.664,388.286,167.548,50.683,159.388
C09775=1021.236,113.914,388.266,167.551,50.678,159.387
C09776=1021.241,114.163,388.247,167.554,50.672,159.386
C09777=1021.247,114.412,388.228,167.557,50.666,159.386
C09778=1021.252,114.661,388.209,167.559,50.660,159.385
C09779=1021.257,114.910,388.190,167.563,50.653,159.384
C09780=1021.263,115.160,388.170,167.566,50.648,159.384
C09781=1021.268,115.408,388.151,167.569,50.642,159.383
C09782=1021.274,115.658,388.132,167.571,50.635,159.382
C09783=1021.279,115.907,388.113,167.574,50.630,159.382
C09784=1021.285,116.156,388.094,167.577,50.624,159.381
C09785=1021.290,116.406,388.075,167.579,50.617,159.380
C09786=1021.295,116.654,388.056,167.583,50.611,159.379
C09787=1021.300,116.904,388.036,167.586,50.605,159.379
C09788=1021.305,117.153,388.017,167.589,50.600,159.378
C09789=1021.311,117.402,387.998,167.591,50.593,159.377
C09790=1021.317,117.652,387.979,167.594,50.587,159.377
C09791=1021.322,117.900,387.960,167.597,50.582,159.376
C09792=1021.328,118.150,387.941,167.599,50.575,159.375
C09793=1021.333,118.399,387.921,167.603,50.569,159.375
C09794=1021.338,118.648,387.902,167.606,50.563,159.374
C09795=1021.344,118.897,387.883,167.609,50.557,159.373
C09796=1021.350,119.147,387.864,167.611,50.551,159.372
C09797=1021.355,119.395,387.845,167.614,50.545,159.372
C09798=1021.360,119.645,387.825,167.618,50.538,159.371
C09799=1021.365,119.895,387.806,167.621,50.533,159.370
C09800=1021.371,120.143,387.787,167.623,50.527,159.370
C09801=1021.376,120.393,387.768,167.626,50.520,159.369
C09802=1021.382,120.642,387.748,167.629,50.514,159.368
C09803=1021.388,120.891,387.729,167.633,50.508,159.368
C09804=1021.393,121.140,387.710,167.635,50.502,159.367
C09805=1021.399,121.389,387.691,167.638,50.496,159.366
C09806=1021.404,121.639,387.671,167.641,50.490,159.365
C09807=1021.409,121.887,387.652,167.643,50.484,159.365
C09808=1021.415,122.137,387.633,167.647,50.478,159.364
C09809=1021.420,122.387,387.613,167.650,50.472,159.363
C09810=1021.426,122.636,387.594,167.652,50.466,159.362
C09811=1021.431,122.884,387.575,167.655,50.460,159.362
C09812=1021.438,123.168,387.552,167.659,50.453,159.361
C09813=1021.444,123.450,387.531,167.662,50.446,159.360
C09814=1021.450,123.733,387.509,167.665,50.439,159.359
C09815=1021.457,124.017,387.487,167.669,50.432,159.359
C09816=1021.462,124.266,387.468,167.672,50.426,159.358
C09817=1021.468,124.515,387.448,167.675,50.419,159.357
C09818=1021.473,124.765,387.429,167.678,50.414,159.357
C09819=1021.479,125.014,387.410,167.680,50.407,159.356
C09820=1021.484,125.263,387.389,167.683,50.401,159.355
C09821=1021.489,125.512,387.371,167.687,50.395,159.354
C09822=1021.495,125.761,387.351,167.690,50.389,159.354
C09823=1021.501,126.011,387.332,167.692,50.383,159.353
C09824=1021.507,126.260,387.312,167.695,50.377,159.352
C09825=1021.512,126.509,387.293,167.699,50.371,159.352
C09826=1021.518,126.758,387.274,167.702,50.365,159.351
C09827=1021.523,127.007,387.255,167.704,50.358,159.350
C09828=1021.529,127.256,387.235,167.708,50.352,159.349
C09829=1021.534,127.506,387.215,167.710,50.346,159.349
C09830=1021.540,127.755,387.196,167.713,50.340,159.348
C09831=1021.545,128.004,387.177,167.716,50.334,159.347
C09832=1021.551,128.253,387.157,167.720,50.328,159.347
C09833=1021.557,128.502,387.138,167.723,50.322,159.346
C09834=1021.562,128.752,387.118,167.725,50.315,159.345
C09835=1021.568,129.000,387.098,167.729,50.309,159.344
C09836=1021.574,129.250,387.079,167.731,50.303,159.344
C09837=1021.579,129.500,387.059,167.734,50.297,159.343
C09838=1021.584,129.748,387.040,167.738,50.290,159.342
C09839=1021.590,129.997,387.021,167.741,50.285,159.341
C09840=1021.596,130.247,387.001,167.744,50.279,159.341
C09841=1021.601,130.496,386.981,167.746,50.272,159.340
C09842=1021.607,130.745,386.961,167.750,50.266,159.339
C09843=1021.612,130.994,386.941,167.753,50.261,159.339
C09844=1021.618,131.244,386.922,167.756,50.255,159.338
C09845=1021.622,131.492,386.901,167.758,50.248,159.337
C09846=1021.628,131.741,386.882,167.762,50.242,159.337
C09847=1021.633,131.991,386.862,167.765,50.237,159.336
C09848=1021.639,132.239,386.842,167.767,50.230,159.335
C09849=1021.645,132.489,386.822,167.770,50.224,159.334
C09850=1021.650,132.738,386.802,167.774,50.218,159.334
C09851=1021.656,132.987,386.783,167.777,50.213,159.333
C09852=1021.661,133.237,386.762,167.780,50.206,159.332
C09853=1021.667,133.486,386.743,167.782,50.201,159.332
C09854=1021.671,133.734,386.723,167.786,50.194,159.331
C09855=1021.677,133.983,386.703,167.789,50.188,159.330
C09856=1021.682,134.233,386.683,167.792,50.182,159.330
C09857=1021.688,134.482,386.663,167.796,50.176,159.329
C09858=1021.694,134.731,386.642,167.798,50.170,159.328
C09859=1021.699,134.980,386.623,167.801,50.164,159.328
C09860=1021.705,135.229,386.603,167.804,50.158,159.327
C09861=1021.710,135.479,386.583,167.808,50.152,159.326
C09862=1021.716,135.728,386.563,167.810,50.146,159.326
C09863=1021.722,135.977,386.543,167.813,50.140,159.325
C09864=1021.726,136.227,386.523,167.817,50.134,159.324
C09865=1021.732,136.475,386.503,167.820,50.128,159.323
C09866=1021.738,136.725,386.482,167.822,50.122,159.323
C09867=1021.744,136.973,386.463,167.825,50.116,159.322
C09868=1021.749,137.223,386.443,167.829,50.110,159.322
C09869=1021.755,137.472,386.423,167.832,50.104,159.321
C09870=1021.760,137.721,386.402,167.835,50.098,159.320
C09871=1021.766,137.970,386.383,167.839,50.092,159.319
C09872=1021.770,138.219,386.363,167.841,50.086,159.319
C09873=1021.776,138.468,386.342,167.844,50.080,159.318
C09874=1021.782,138.717,386.322,167.848,50.074,159.317
C09875=1021.787,138.966,386.302,167.851,50.068,159.317
C09876=1021.793,139.250,386.279,167.854,50.061,159.316
C09877=1021.799,139.533,386.256,167.858,50.055,159.315
C09878=1021.805,139.816,386.232,167.861,50.048,159.314
C09879=1021.812,140.099,386.209,167.865,50.041,159.314
C09880=1021.817,140.348,386.189,167.868,50.035,159.313
C09881=1021.822,140.597,386.168,167.870,50.029,159.312
C09882=1021.827,140.847,386.148,167.874,50.023,159.312
C09883=1021.833,141.095,386.129,167.877,50.017,159.311
C09884=1021.839,141.344,386.108,167.880,50.011,159.310
C09885=1021.844,141.594,386.087,167.884,50.005,159.310
C09886=1021.850,141.842,386.067,167.887,49.999,159.309
C09887=1021.855,142.092,386.047,167.890,49.994,159.308
C09888=1021.860,142.341,386.026,167.893,49.987,159.307
C09889=1021.866,142.590,386.006,167.896,49.981,159.307
C09890=1021.872,142.839,385.986,167.899,49.975,159.306
C09891=1021.877,143.088,385.965,167.903,49.969,159.306
C09892=1021.882,143.337,385.945,167.905,49.963,159.305
C09893=1021.887,143.586,385.924,167.908,49.957,159.304
C09894=1021.893,143.835,385.904,167.912,49.951,159.303
C09895=1021.899,144.085,385.883,167.915,49.946,159.303
C09896=1021.904,144.334,385.863,167.918,49.940,159.302
C09897=1021.910,144.583,385.842,167.922,49.933,159.301
C09898=1021.916,144.832,385.822,167.924,49.928,159.301
C09899=1021.921,145.081,385.802,167.927,49.922,159.300
C09900=1021.926,145.330,385.781,167.931,49.915,159.299
C09901=1021.931,145.579,385.761,167.934,49.909,159.299
C09902=1021.937,145.828,385.741,167.937,49.904,159.298
C09903=1021.943,146.077,385.720,167.941,49.898,159.297
C09904=1021.948,146.326,385.699,167.944,49.892,159.297
C09905=1021.954,146.576,385.679,167.946,49.886,159.296
C09906=1021.959,146.825,385.658,167.950,49.880,159.295
C09907=1021.965,147.074,385.637,167.953,49.874,159.295
C09908=1021.970,147.323,385.616,167.957,49.868,159.294
C09909=1021.975,147.572,385.596,167.960,49.862,159.293
C09910=1021.980,147.821,385.575,167.963,49.857,159.293
C09911=1021.986,148.070,385.555,167.966,49.850,159.292
C09912=1021.991,148.319,385.533,167.969,49.844,159.291
C09913=1021.997,148.568,385.512,167.972,49.839,159.291
C09914=1022.002,148.818,385.492,167.976,49.833,159.290
C09915=1022.008,149.067,385.471,167.979,49.827,159.289
C09916=1022.013,149.315,385.450,167.982,49.821,159.289
C09917=1022.018,149.564,385.429,167.986,49.815,159.288
C09918=1022.024,149.813,385.409,167.988,49.809,159.287
C09919=1022.029,150.063,385.388,167.991,49.803,159.287
C09920=1022.035,150.312,385.367,167.995,49.797,159.286
C09921=1022.040,150.561,385.346,167.998,49.791,159.285
C09922=1022.046,150.810,385.326,168.002,49.785,159.285
C09923=1022.051,151.058,385.304,168.005,49.780,159.284
C09924=1022.056,151.308,385.284,168.008,49.773,159.283
C09925=1022.062,151.557,385.263,168.012,49.767,159.283
C09926=1022.068,151.806,385.242,168.015,49.762,159.282
C09927=1022.073,152.055,385.221,168.018,49.756,159.281
C09928=1022.078,152.304,385.200,168.021,49.750,159.281
C09929=1022.084,152.553,385.179,168.024,49.744,159.280
C09930=1022.090,152.803,385.158,168.028,49.738,159.280
C09931=1022.095,153.052,385.138,168.031,49.732,159.279
C09932=1022.101,153.348,385.112,168.035,49.725,159.278
C09933=1022.108,153.646,385.088,168.039,49.718,159.277
C09934=1022.114,153.942,385.062,168.043,49.712,159.277
C09935=1022.121,154.239,385.037,168.047,49.704,159.276
C09936=1022.127,154.482,385.017,168.050,49.698,159.275
C09937=1022.132,154.723,384.996,168.053,49.693,159.274
C09938=1022.136,154.965,384.976,168.056,49.688,159.274
C09939=1022.142,155.206,384.955,168.060,49.682,159.273
C09940=1022.147,155.449,384.935,168.063,49.676,159.273
C09941=1022.153,155.691,384.914,168.066,49.671,159.272
C09942=1022.157,155.933,384.893,168.069,49.665,159.271
C09943=1022.164,156.175,384.873,168.073,49.659,159.271
C09944=1022.169,156.424,384.852,168.076,49.653,159.270
C09945=1022.174,156.673,384.830,168.080,49.647,159.270
C09946=1022.179,156.922,384.809,168.083,49.642,159.269
C09947=1022.185,157.171,384.788,168.085,49.635,159.268
C09948=1022.190,157.420,384.768,168.089,49.629,159.267
C09949=1022.196,157.669,384.746,168.092,49.624,159.267
C09950=1022.201,157.919,384.725,168.096,49.618,159.266
C09951=1022.207,158.167,384.704,168.099,49.612,159.266
C09952=1022.213,158.416,384.682,168.103,49.606,159.265
C09953=1022.218,158.665,384.661,168.106,49.600,159.264
C09954=1022.223,158.914,384.640,168.110,49.594,159.264
C09955=1022.229,159.164,384.618,168.113,49.589,159.263
C09956=1022.234,159.413,384.597,168.116,49.583,159.262
C09957=1022.239,159.661,384.575,168.120,49.577,159.262
C09958=1022.244,159.911,384.553,168.123,49.572,159.261
C09959=1022.250,160.159,384.532,168.126,49.566,159.260
C09960=1022.255,160.408,384.510,168.130,49.560,159.260
C09961=1022.260,160.658,384.488,168.133,49.555,159.259
C09962=1022.266,160.906,384.467,168.136,49.549,159.259
C09963=1022.270,161.156,384.445,168.140,49.543,159.258
C09964=1022.276,161.405,384.424,168.143,49.538,159.258
C09965=1022.281,161.654,384.402,168.147,49.532,159.257
C09966=1022.286,161.903,384.380,168.150,49.526,159.256
C09967=1022.292,162.152,384.358,168.153,49.521,159.256
C09968=1022.297,162.401,384.337,168.157,49.515,159.255
C09969=1022.302,162.649,384.315,168.160,49.510,159.255
C09970=1022.308,162.899,384.293,168.164,49.504,159.254
C09971=1022.313,163.147,384.271,168.167,49.498,159.253
C09972=1022.318,163.396,384.249,168.170,49.492,159.253
C09973=1022.324,163.645,384.228,168.174,49.487,159.252
C09974=1022.329,163.894,384.206,168.177,49.481,159.251
C09975=1022.334,164.144,384.184,168.181,49.475,159.251
C09976=1022.340,164.392,384.162,168.184,49.469,159.250
C09977=1022.345,164.641,384.140,168.187,49.464,159.249
C09978=1022.350,164.891,384.118,168.191,49.458,159.249
C09979=1022.356,165.139,384.097,168.194,49.453,159.248
C09980=1022.361,165.389,384.075,168.198,49.447,159.248
C09981=1022.367,165.637,384.053,168.201,49.441,159.247
C09982=1022.371,165.886,384.032,168.205,49.435,159.247
C09983=1022.377,166.135,384.009,168.208,49.430,159.246
C09984=1022.382,166.384,383.988,168.212,49.424,159.245
C09985=1022.388,166.634,383.966,168.215,49.418,159.245
C09986=1022.393,166.882,383.944,168.218,49.412,159.244
C09987=1022.399,167.132,383.922,168.223,49.407,159.244
C09988=1022.404,167.380,383.901,168.225,49.402,159.243
C09989=1022.409,167.630,383.878,168.229,49.396,159.242
C09990=1022.415,167.878,383.857,168.232,49.390,159.242
C09991=1022.420,168.128,383.835,168.236,49.384,159.241
C09992=1022.425,168.376,383.812,168.239,49.379,159.240
C09993=1022.431,168.625,383.791,168.243,49.373,159.240
C09994=1022.436,168.874,383.769,168.246,49.367,159.239
C09995=1022.441,169.124,383.746,168.250,49.361,159.239
C09996=1022.447,169.372,383.725,168.253,49.355,159.238
//INST
///DATE 2021/06/25 14:49
///ATTR SC,RW,RJ
////FRAME ROBOT
///GROUP1 RB1
NOP
MOVL C00000 V=800.0 PL=0
MOVL C00001 V=800.0 PL=0
MOVL C00002 V=800.0 PL=0
MOVL C00003 V=800.0 PL=0
MOVL C00004 V=800.0 PL=0
MOVL C00005 V=800.0 PL=0
MOVL C00006 V=800.0 PL=0
MOVL C00007 V=800.0 PL=0
MOVL C00008 V=800.0 PL=0
MOVL C00009 V=800.0 PL=0
MOVL C00010 V=800.0 PL=0
MOVL C00011 V=800.0 PL=0
MOVL C00012 V=800.0 PL=0
MOVL C00013 V=800.0 PL=0
MOVL C00014 V=800.0 PL=0
MOVL C00015 V=800.0 PL=0
MOVL C00016 V=800.0 PL=0
MOVL C00017 V=800.0 PL=0
MOVL C00018 V=800.0 PL=0
MOVL C00019 V=800.0 PL=0
MOVL C00020 V=800.0 PL=0
MOVL C00021 V=800.0 PL=0
MOVL C00022 V=800.0 PL=0
MOVL C00023 V=800.0 PL=0
MOVL C00024 V=800.0 PL=0
MOVL C00025 V=800.0 PL=0
MOVL C00026 V=800.0 PL=0
MOVL C00027 V=800.0 PL=0
MOVL C00028 V=800.0 PL=0
MOVL C00029 V=800.0 PL=0
MOVL C00030 V=800.0 PL=0
MOVL C00031 V=800.0 PL=0
MOVL C00032 V=800.0 PL=0
MOVL C00033 V=800.0 PL=0
MOVL C00034 V=800.0 PL=0
MOVL C00035 V=800.0 PL=0
MOVL C00036 V=800.0 PL=0
MOVL C00037 V=800.0 PL=0
MOVL C00038 V=800.0 PL=0
MOVL C00039 V=800.0 PL=0
MOVL C00040 V=800.0 PL=0
MOVL C00041 V=800.0 PL=0
MOVL C00042 V=800.0 PL=0
MOVL C00043 V=800.0 PL=0
MOVL C00044 V=800.0 PL=0
MOVL C00045 V=800.0 PL=0
MOVL C00046 V=800.0 PL=0
MOVL C00047 V=800.0 PL=0
MOVL C00048 V=800.0 PL=0
MOVL C00049 V=800.0 PL=0
MOVL C00050 V=800.0 PL=0
MOVL C00051 V=800.0 PL=0
MOVL C00052 V=800.0 PL=0
MOVL C00053 V=800.0 PL=0
MOVL C00054 V=800.0 PL=0
MOVL C00055 V=800.0 PL=0
MOVL C00056 V=800.0 PL=0
MOVL C00057 V=800.0 PL=0
MOVL C00058 V=800.0 PL=0
MOVL C00059 V=800.0 PL=0
MOVL C00060 V=800.0 PL=0
MOVL C00061 V=800.0 PL=0
MOVL C00062 V=800.0 PL=0
MOVL C00063 V=800.0 PL=0
MOVL C00064 V=800.0 PL=0
MOVL C00065 V=800.0 PL=0
MOVL C00066 V=800.0 PL=0
MOVL C00067 V=800.0 PL=0
MOVL C00068 V=800.0 PL=0
MOVL C00069 V=800.0 PL=0
MOVL C00070 V=800.0 PL=0
MOVL C00071 V=800.0 PL=0
MOVL C00072 V=800.0 PL=0
MOVL C00073 V=800.0 PL=0
MOVL C00074 V=800.0 PL=0
MOVL C00075 V=800.0 PL=0
MOVL C00076 V=800.0 PL=0
MOVL C00077 V=800.0 PL=0
MOVL C00078 V=800.0 PL=0
MOVL C00079 V=800.0 PL=0
MOVL C00080 V=800.0 PL=0
MOVL C00081 V=800.0 PL=0
MOVL C00082 V=800.0 PL=0
MOVL C00083 V=800.0 PL=0
MOVL C00084 V=800.0 PL=0
MOVL C00085 V=800.0 PL=0
MOVL C00086 V=800.0 PL=0
MOVL C00087 V=800.0 PL=0
MOVL C00088 V=800.0 PL=0
MOVL C00089 V=800.0 PL=0
MOVL C00090 V=800.0 PL=0
MOVL C00091 V=800.0 PL=0
MOVL C00092 V=800.0 PL=0
MOVL C00093 V=800.0 PL=0
MOVL C00094 V=800.0 PL=0
MOVL C00095 V=800.0 PL=0
MOVL C00096 V=800.0 PL=0
MOVL C00097 V=800.0 PL=0
MOVL C00098 V=800.0 PL=0
MOVL C00099 V=800.0 PL=0
MOVL C00100 V=800.0 PL=0
MOVL C00101 V=800.0 PL=0
MOVL C00102 V=800.0 PL=0
MOVL C00103 V=800.0 PL=0
MOVL C00104 V=800.0 PL=0
MOVL C00105 V=800.0 PL=0
MOVL C00106 V=800.0 PL=0
MOVL C00107 V=800.0 PL=0
MOVL C00108 V=800.0 PL=0
MOVL C00109 V=800.0 PL=0
MOVL C00110 V=800.0 PL=0
MOVL C00111 V=800.0 PL=0
MOVL C00112 V=800.0 PL=0
MOVL C00113 V=800.0 PL=0
MOVL C00114 V=800.0 PL=0
MOVL C00115 V=800.0 PL=0
MOVL C00116 V=800.0 PL=0
MOVL C00117 V=800.0 PL=0
MOVL C00118 V=800.0 PL=0
MOVL C00119 V=800.0 PL=0
MOVL C00120 V=800.0 PL=0
MOVL C00121 V=800.0 PL=0
MOVL C00122 V=800.0 PL=0
MOVL C00123 V=800.0 PL=0
MOVL C00124 V=800.0 PL=0
MOVL C00125 V=800.0 PL=0
MOVL C00126 V=800.0 PL=0
MOVL C00127 V=800.0 PL=0
MOVL C00128 V=800.0 PL=0
MOVL C00129 V=800.0 PL=0
MOVL C00130 V=800.0 PL=0
MOVL C00131 V=800.0 PL=0
MOVL C00132 V=800.0 PL=0
MOVL C00133 V=800.0 PL=0
MOVL C00134 V=800.0 PL=0
MOVL C00135 V=800.0 PL=0
MOVL C00136 V=800.0 PL=0
MOVL C00137 V=800.0 PL=0
MOVL C00138 V=800.0 PL=0
MOVL C00139 V=800.0 PL=0
MOVL C00140 V=800.0 PL=0
MOVL C00141 V=800.0 PL=0
MOVL C00142 V=800.0 PL=0
MOVL C00143 V=800.0 PL=0
MOVL C00144 V=800.0 PL=0
MOVL C00145 V=800.0 PL=0
MOVL C00146 V=800.0 PL=0
MOVL C00147 V=800.0 PL=0
MOVL C00148 V=800.0 PL=0
MOVL C00149 V=800.0 PL=0
MOVL C00150 V=800.0 PL=0
MOVL C00151 V=800.0 PL=0
MOVL C00152 V=800.0 PL=0
MOVL C00153 V=800.0 PL=0
MOVL C00154 V=800.0 PL=0
MOVL C00155 V=800.0 PL=0
MOVL C00156 V=800.0 PL=0
MOVL C00157 V=800.0 PL=0
MOVL C00158 V=800.0 PL=0
MOVL C00159 V=800.0 PL=0
MOVL C00160 V=800.0 PL=0
MOVL C00161 V=800.0 PL=0
MOVL C00162 V=800.0 PL=0
MOVL C00163 V=800.0 PL=0
MOVL C00164 V=800.0 PL=0
MOVL C00165 V=800.0 PL=0
MOVL C00166 V=800.0 PL=0
MOVL C00167 V=800.0 PL=0
MOVL C00168 V=800.0 PL=0
MOVL C00169 V=800.0 PL=0
MOVL C00170 V=800.0 PL=0
MOVL C00171 V=800.0 PL=0
MOVL C00172 V=800.0 PL=0
MOVL C00173 V=800.0 PL=0
MOVL C00174 V=800.0 PL=0
MOVL C00175 V=800.0 PL=0
MOVL C00176 V=800.0 PL=0
MOVL C00177 V=800.0 PL=0
MOVL C00178 V=800.0 PL=0
MOVL C00179 V=800.0 PL=0
MOVL C00180 V=800.0 PL=0
MOVL C00181 V=800.0 PL=0
MOVL C00182 V=800.0 PL=0
MOVL C00183 V=800.0 PL=0
MOVL C00184 V=800.0 PL=0
MOVL C00185 V=800.0 PL=0
MOVL C00186 V=800.0 PL=0
MOVL C00187 V=800.0 PL=0
MOVL C00188 V=800.0 PL=0
MOVL C00189 V=800.0 PL=0
MOVL C00190 V=800.0 PL=0
MOVL C00191 V=800.0 PL=0
MOVL C00192 V=800.0 PL=0
MOVL C00193 V=800.0 PL=0
MOVL C00194 V=800.0 PL=0
MOVL C00195 V=800.0 PL=0
MOVL C00196 V=800.0 PL=0
MOVL C00197 V=800.0 PL=0
MOVL C00198 V=800.0 PL=0
MOVL C00199 V=800.0 PL=0
MOVL C00200 V=800.0 PL=0
MOVL C00201 V=800.0 PL=0
MOVL C00202 V=800.0 PL=0
MOVL C00203 V=800.0 PL=0
MOVL C00204 V=800.0 PL=0
MOVL C00205 V=800.0 PL=0
MOVL C00206 V=800.0 PL=0
MOVL C00207 V=800.0 PL=0
MOVL C00208 V=800.0 PL=0
MOVL C00209 V=800.0 PL=0
MOVL C00210 V=800.0 PL=0
MOVL C00211 V=800.0 PL=0
MOVL C00212 V=800.0 PL=0
MOVL C00213 V=800.0 PL=0
MOVL C00214 V=800.0 PL=0
MOVL C00215 V=800.0 PL=0
MOVL C00216 V=800.0 PL=0
MOVL C00217 V=800.0 PL=0
MOVL C00218 V=800.0 PL=0
MOVL C00219 V=800.0 PL=0
MOVL C00220 V=800.0 PL=0
MOVL C00221 V=800.0 PL=0
MOVL C00222 V=800.0 PL=0
MOVL C00223 V=800.0 PL=0
MOVL C00224 V=800.0 PL=0
MOVL C00225 V=800.0 PL=0
MOVL C00226 V=800.0 PL=0
MOVL C00227 V=800.0 PL=0
MOVL C00228 V=800.0 PL=0
MOVL C00229 V=800.0 PL=0
MOVL C00230 V=800.0 PL=0
MOVL C00231 V=800.0 PL=0
MOVL C00232 V=800.0 PL=0
MOVL C00233 V=800.0 PL=0
MOVL C00234 V=800.0 PL=0
MOVL C00235 V=800.0 PL=0
MOVL C00236 V=800.0 PL=0
MOVL C00237 V=800.0 PL=0
MOVL C00238 V=800.0 PL=0
MOVL C00239 V=800.0 PL=0
MOVL C00240 V=800.0 PL=0
MOVL C00241 V=800.0 PL=0
MOVL C00242 V=800.0 PL=0
MOVL C00243 V=800.0 PL=0
MOVL C00244 V=800.0 PL=0
MOVL C00245 V=800.0 PL=0
MOVL C00246 V=800.0 PL=0
MOVL C00247 V=800.0 PL=0
MOVL C00248 V=800.0 PL=0
MOVL C00249 V=800.0 PL=0
MOVL C00250 V=800.0 PL=0
MOVL C00251 V=800.0 PL=0
MOVL C00252 V=800.0 PL=0
MOVL C00253 V=800.0 PL=0
MOVL C00254 V=800.0 PL=0
MOVL C00255 V=800.0 PL=0
MOVL C00256 V=800.0 PL=0
MOVL C00257 V=800.0 PL=0
MOVL C00258 V=800.0 PL=0
MOVL C00259 V=800.0 PL=0
MOVL C00260 V=800.0 PL=0
MOVL C00261 V=800.0 PL=0
MOVL C00262 V=800.0 PL=0
MOVL C00263 V=800.0 PL=0
MOVL C00264 V=800.0 PL=0
MOVL C00265 V=800.0 PL=0
MOVL C00266 V=800.0 PL=0
MOVL C00267 V=800.0 PL=0
MOVL C00268 V=800.0 PL=0
MOVL C00269 V=800.0 PL=0
MOVL C00270 V=800.0 PL=0
MOVL C00271 V=800.0 PL=0
MOVL C00272 V=800.0 PL=0
MOVL C00273 V=800.0 PL=0
MOVL C00274 V=800.0 PL=0
MOVL C00275 V=800.0 PL=0
MOVL C00276 V=800.0 PL=0
MOVL C00277 V=800.0 PL=0
MOVL C00278 V=800.0 PL=0
MOVL C00279 V=800.0 PL=0
MOVL C00280 V=800.0 PL=0
MOVL C00281 V=800.0 PL=0
MOVL C00282 V=800.0 PL=0
MOVL C00283 V=800.0 PL=0
MOVL C00284 V=800.0 PL=0
MOVL C00285 V=800.0 PL=0
MOVL C00286 V=800.0 PL=0
MOVL C00287 V=800.0 PL=0
MOVL C00288 V=800.0 PL=0
MOVL C00289 V=800.0 PL=0
MOVL C00290 V=800.0 PL=0
MOVL C00291 V=800.0 PL=0
MOVL C00292 V=800.0 PL=0
MOVL C00293 V=800.0 PL=0
MOVL C00294 V=800.0 PL=0
MOVL C00295 V=800.0 PL=0
MOVL C00296 V=800.0 PL=0
MOVL C00297 V=800.0 PL=0
MOVL C00298 V=800.0 PL=0
MOVL C00299 V=800.0 PL=0
MOVL C00300 V=800.0 PL=0
MOVL C00301 V=800.0 PL=0
MOVL C00302 V=800.0 PL=0
MOVL C00303 V=800.0 PL=0
MOVL C00304 V=800.0 PL=0
MOVL C00305 V=800.0 PL=0
MOVL C00306 V=800.0 PL=0
MOVL C00307 V=800.0 PL=0
MOVL C00308 V=800.0 PL=0
MOVL C00309 V=800.0 PL=0
MOVL C00310 V=800.0 PL=0
MOVL C00311 V=800.0 PL=0
MOVL C00312 V=800.0 PL=0
MOVL C00313 V=800.0 PL=0
MOVL C00314 V=800.0 PL=0
MOVL C00315 V=800.0 PL=0
MOVL C00316 V=800.0 PL=0
MOVL C00317 V=800.0 PL=0
MOVL C00318 V=800.0 PL=0
MOVL C00319 V=800.0 PL=0
MOVL C00320 V=800.0 PL=0
MOVL C00321 V=800.0 PL=0
MOVL C00322 V=800.0 PL=0
MOVL C00323 V=800.0 PL=0
MOVL C00324 V=800.0 PL=0
MOVL C00325 V=800.0 PL=0
MOVL C00326 V=800.0 PL=0
MOVL C00327 V=800.0 PL=0
MOVL C00328 V=800.0 PL=0
MOVL C00329 V=800.0 PL=0
MOVL C00330 V=800.0 PL=0
MOVL C00331 V=800.0 PL=0
MOVL C00332 V=800.0 PL=0
MOVL C00333 V=800.0 PL=0
MOVL C00334 V=800.0 PL=0
MOVL C00335 V=800.0 PL=0
MOVL C00336 V=800.0 PL=0
MOVL C00337 V=800.0 PL=0
MOVL C00338 V=800.0 PL=0
MOVL C00339 V=800.0 PL=0
MOVL C00340 V=800.0 PL=0
MOVL C00341 V=800.0 PL=0
MOVL C00342 V=800.0 PL=0
MOVL C00343 V=800.0 PL=0
MOVL C00344 V=800.0 PL=0
MOVL C00345 V=800.0 PL=0
MOVL C00346 V=800.0 PL=0
MOVL C00347 V=800.0 PL=0
MOVL C00348 V=800.0 PL=0
MOVL C00349 V=800.0 PL=0
MOVL C00350 V=800.0 PL=0
MOVL C00351 V=800.0 PL=0
MOVL C00352 V=800.0 PL=0
MOVL C00353 V=800.0 PL=0
MOVL C00354 V=800.0 PL=0
MOVL C00355 V=800.0 PL=0
MOVL C00356 V=800.0 PL=0
MOVL C00357 V=800.0 PL=0
MOVL C00358 V=800.0 PL=0
MOVL C00359 V=800.0 PL=0
MOVL C00360 V=800.0 PL=0
MOVL C00361 V=800.0 PL=0
MOVL C00362 V=800.0 PL=0
MOVL C00363 V=800.0 PL=0
MOVL C00364 V=800.0 PL=0
MOVL C00365 V=800.0 PL=0
MOVL C00366 V=800.0 PL=0
MOVL C00367 V=800.0 PL=0
MOVL C00368 V=800.0 PL=0
MOVL C00369 V=800.0 PL=0
MOVL C00370 V=800.0 PL=0
MOVL C00371 V=800.0 PL=0
MOVL C00372 V=800.0 PL=0
MOVL C00373 V=800.0 PL=0
MOVL C00374 V=800.0 PL=0
MOVL C00375 V=800.0 PL=0
MOVL C00376 V=800.0 PL=0
MOVL C00377 V=800.0 PL=0
MOVL C00378 V=800.0 PL=0
MOVL C00379 V=800.0 PL=0
MOVL C00380 V=800.0 PL=0
MOVL C00381 V=800.0 PL=0
MOVL C00382 V=800.0 PL=0
MOVL C00383 V=800.0 PL=0
MOVL C00384 V=800.0 PL=0
MOVL C00385 V=800.0 PL=0
MOVL C00386 V=800.0 PL=0
MOVL C00387 V=800.0 PL=0
MOVL C00388 V=800.0 PL=0
MOVL C00389 V=800.0 PL=0
MOVL C00390 V=800.0 PL=0
MOVL C00391 V=800.0 PL=0
MOVL C00392 V=800.0 PL=0
MOVL C00393 V=800.0 PL=0
MOVL C00394 V=800.0 PL=0
MOVL C00395 V=800.0 PL=0
MOVL C00396 V=800.0 PL=0
MOVL C00397 V=800.0 PL=0
MOVL C00398 V=800.0 PL=0
MOVL C00399 V=800.0 PL=0
MOVL C00400 V=800.0 PL=0
MOVL C00401 V=800.0 PL=0
MOVL C00402 V=800.0 PL=0
MOVL C00403 V=800.0 PL=0
MOVL C00404 V=800.0 PL=0
MOVL C00405 V=800.0 PL=0
MOVL C00406 V=800.0 PL=0
MOVL C00407 V=800.0 PL=0
MOVL C00408 V=800.0 PL=0
MOVL C00409 V=800.0 PL=0
MOVL C00410 V=800.0 PL=0
MOVL C00411 V=800.0 PL=0
MOVL C00412 V=800.0 PL=0
MOVL C00413 V=800.0 PL=0
MOVL C00414 V=800.0 PL=0
MOVL C00415 V=800.0 PL=0
MOVL C00416 V=800.0 PL=0
MOVL C00417 V=800.0 PL=0
MOVL C00418 V=800.0 PL=0
MOVL C00419 V=800.0 PL=0
MOVL C00420 V=800.0 PL=0
MOVL C00421 V=800.0 PL=0
MOVL C00422 V=800.0 PL=0
MOVL C00423 V=800.0 PL=0
MOVL C00424 V=800.0 PL=0
MOVL C00425 V=800.0 PL=0
MOVL C00426 V=800.0 PL=0
MOVL C00427 V=800.0 PL=0
MOVL C00428 V=800.0 PL=0
MOVL C00429 V=800.0 PL=0
MOVL C00430 V=800.0 PL=0
MOVL C00431 V=800.0 PL=0
MOVL C00432 V=800.0 PL=0
MOVL C00433 V=800.0 PL=0
MOVL C00434 V=800.0 PL=0
MOVL C00435 V=800.0 PL=0
MOVL C00436 V=800.0 PL=0
MOVL C00437 V=800.0 PL=0
MOVL C00438 V=800.0 PL=0
MOVL C00439 V=800.0 PL=0
MOVL C00440 V=800.0 PL=0
MOVL C00441 V=800.0 PL=0
MOVL C00442 V=800.0 PL=0
MOVL C00443 V=800.0 PL=0
MOVL C00444 V=800.0 PL=0
MOVL C00445 V=800.0 PL=0
MOVL C00446 V=800.0 PL=0
MOVL C00447 V=800.0 PL=0
MOVL C00448 V=800.0 PL=0
MOVL C00449 V=800.0 PL=0
MOVL C00450 V=800.0 PL=0
MOVL C00451 V=800.0 PL=0
MOVL C00452 V=800.0 PL=0
MOVL C00453 V=800.0 PL=0
MOVL C00454 V=800.0 PL=0
MOVL C00455 V=800.0 PL=0
MOVL C00456 V=800.0 PL=0
MOVL C00457 V=800.0 PL=0
MOVL C00458 V=800.0 PL=0
MOVL C00459 V=800.0 PL=0
MOVL C00460 V=800.0 PL=0
MOVL C00461 V=800.0 PL=0
MOVL C00462 V=800.0 PL=0
MOVL C00463 V=800.0 PL=0
MOVL C00464 V=800.0 PL=0
MOVL C00465 V=800.0 PL=0
MOVL C00466 V=800.0 PL=0
MOVL C00467 V=800.0 PL=0
MOVL C00468 V=800.0 PL=0
MOVL C00469 V=800.0 PL=0
MOVL C00470 V=800.0 PL=0
MOVL C00471 V=800.0 PL=0
MOVL C00472 V=800.0 PL=0
MOVL C00473 V=800.0 PL=0
MOVL C00474 V=800.0 PL=0
MOVL C00475 V=800.0 PL=0
MOVL C00476 V=800.0 PL=0
MOVL C00477 V=800.0 PL=0
MOVL C00478 V=800.0 PL=0
MOVL C00479 V=800.0 PL=0
MOVL C00480 V=800.0 PL=0
MOVL C00481 V=800.0 PL=0
MOVL C00482 V=800.0 PL=0
MOVL C00483 V=800.0 PL=0
MOVL C00484 V=800.0 PL=0
MOVL C00485 V=800.0 PL=0
MOVL C00486 V=800.0 PL=0
MOVL C00487 V=800.0 PL=0
MOVL C00488 V=800.0 PL=0
MOVL C00489 V=800.0 PL=0
MOVL C00490 V=800.0 PL=0
MOVL C00491 V=800.0 PL=0
MOVL C00492 V=800.0 PL=0
MOVL C00493 V=800.0 PL=0
MOVL C00494 V=800.0 PL=0
MOVL C00495 V=800.0 PL=0
MOVL C00496 V=800.0 PL=0
MOVL C00497 V=800.0 PL=0
MOVL C00498 V=800.0 PL=0
MOVL C00499 V=800.0 PL=0
MOVL C00500 V=800.0 PL=0
MOVL C00501 V=800.0 PL=0
MOVL C00502 V=800.0 PL=0
MOVL C00503 V=800.0 PL=0
MOVL C00504 V=800.0 PL=0
MOVL C00505 V=800.0 PL=0
MOVL C00506 V=800.0 PL=0
MOVL C00507 V=800.0 PL=0
MOVL C00508 V=800.0 PL=0
MOVL C00509 V=800.0 PL=0
MOVL C00510 V=800.0 PL=0
MOVL C00511 V=800.0 PL=0
MOVL C00512 V=800.0 PL=0
MOVL C00513 V=800.0 PL=0
MOVL C00514 V=800.0 PL=0
MOVL C00515 V=800.0 PL=0
MOVL C00516 V=800.0 PL=0
MOVL C00517 V=800.0 PL=0
MOVL C00518 V=800.0 PL=0
MOVL C00519 V=800.0 PL=0
MOVL C00520 V=800.0 PL=0
MOVL C00521 V=800.0 PL=0
MOVL C00522 V=800.0 PL=0
MOVL C00523 V=800.0 PL=0
MOVL C00524 V=800.0 PL=0
MOVL C00525 V=800.0 PL=0
MOVL C00526 V=800.0 PL=0
MOVL C00527 V=800.0 PL=0
MOVL C00528 V=800.0 PL=0
MOVL C00529 V=800.0 PL=0
MOVL C00530 V=800.0 PL=0
MOVL C00531 V=800.0 PL=0
MOVL C00532 V=800.0 PL=0
MOVL C00533 V=800.0 PL=0
MOVL C00534 V=800.0 PL=0
MOVL C00535 V=800.0 PL=0
MOVL C00536 V=800.0 PL=0
MOVL C00537 V=800.0 PL=0
MOVL C00538 V=800.0 PL=0
MOVL C00539 V=800.0 PL=0
MOVL C00540 V=800.0 PL=0
MOVL C00541 V=800.0 PL=0
MOVL C00542 V=800.0 PL=0
MOVL C00543 V=800.0 PL=0
MOVL C00544 V=800.0 PL=0
MOVL C00545 V=800.0 PL=0
MOVL C00546 V=800.0 PL=0
MOVL C00547 V=800.0 PL=0
MOVL C00548 V=800.0 PL=0
MOVL C00549 V=800.0 PL=0
MOVL C00550 V=800.0 PL=0
MOVL C00551 V=800.0 PL=0
MOVL C00552 V=800.0 PL=0
MOVL C00553 V=800.0 PL=0
MOVL C00554 V=800.0 PL=0
MOVL C00555 V=800.0 PL=0
MOVL C00556 V=800.0 PL=0
MOVL C00557 V=800.0 PL=0
MOVL C00558 V=800.0 PL=0
MOVL C00559 V=800.0 PL=0
MOVL C00560 V=800.0 PL=0
MOVL C00561 V=800.0 PL=0
MOVL C00562 V=800.0 PL=0
MOVL C00563 V=800.0 PL=0
MOVL C00564 V=800.0 PL=0
MOVL C00565 V=800.0 PL=0
MOVL C00566 V=800.0 PL=0
MOVL C00567 V=800.0 PL=0
MOVL C00568 V=800.0 PL=0
MOVL C00569 V=800.0 PL=0
MOVL C00570 V=800.0 PL=0
MOVL C00571 V=800.0 PL=0
MOVL C00572 V=800.0 PL=0
MOVL C00573 V=800.0 PL=0
MOVL C00574 V=800.0 PL=0
MOVL C00575 V=800.0 PL=0
MOVL C00576 V=800.0 PL=0
MOVL C00577 V=800.0 PL=0
MOVL C00578 V=800.0 PL=0
MOVL C00579 V=800.0 PL=0
MOVL C00580 V=800.0 PL=0
MOVL C00581 V=800.0 PL=0
MOVL C00582 V=800.0 PL=0
MOVL C00583 V=800.0 PL=0
MOVL C00584 V=800.0 PL=0
MOVL C00585 V=800.0 PL=0
MOVL C00586 V=800.0 PL=0
MOVL C00587 V=800.0 PL=0
MOVL C00588 V=800.0 PL=0
MOVL C00589 V=800.0 PL=0
MOVL C00590 V=800.0 PL=0
MOVL C00591 V=800.0 PL=0
MOVL C00592 V=800.0 PL=0
MOVL C00593 V=800.0 PL=0
MOVL C00594 V=800.0 PL=0
MOVL C00595 V=800.0 PL=0
MOVL C00596 V=800.0 PL=0
MOVL C00597 V=800.0 PL=0
MOVL C00598 V=800.0 PL=0
MOVL C00599 V=800.0 PL=0
MOVL C00600 V=800.0 PL=0
MOVL C00601 V=800.0 PL=0
MOVL C00602 V=800.0 PL=0
MOVL C00603 V=800.0 PL=0
MOVL C00604 V=800.0 PL=0
MOVL C00605 V=800.0 PL=0
MOVL C00606 V=800.0 PL=0
MOVL C00607 V=800.0 PL=0
MOVL C00608 V=800.0 PL=0
MOVL C00609 V=800.0 PL=0
MOVL C00610 V=800.0 PL=0
MOVL C00611 V=800.0 PL=0
MOVL C00612 V=800.0 PL=0
MOVL C00613 V=800.0 PL=0
MOVL C00614 V=800.0 PL=0
MOVL C00615 V=800.0 PL=0
MOVL C00616 V=800.0 PL=0
MOVL C00617 V=800.0 PL=0
MOVL C00618 V=800.0 PL=0
MOVL C00619 V=800.0 PL=0
MOVL C00620 V=800.0 PL=0
MOVL C00621 V=800.0 PL=0
MOVL C00622 V=800.0 PL=0
MOVL C00623 V=800.0 PL=0
MOVL C00624 V=800.0 PL=0
MOVL C00625 V=800.0 PL=0
MOVL C00626 V=800.0 PL=0
MOVL C00627 V=800.0 PL=0
MOVL C00628 V=800.0 PL=0
MOVL C00629 V=800.0 PL=0
MOVL C00630 V=800.0 PL=0
MOVL C00631 V=800.0 PL=0
MOVL C00632 V=800.0 PL=0
MOVL C00633 V=800.0 PL=0
MOVL C00634 V=800.0 PL=0
MOVL C00635 V=800.0 PL=0
MOVL C00636 V=800.0 PL=0
MOVL C00637 V=800.0 PL=0
MOVL C00638 V=800.0 PL=0
MOVL C00639 V=800.0 PL=0
MOVL C00640 V=800.0 PL=0
MOVL C00641 V=800.0 PL=0
MOVL C00642 V=800.0 PL=0
MOVL C00643 V=800.0 PL=0
MOVL C00644 V=800.0 PL=0
MOVL C00645 V=800.0 PL=0
MOVL C00646 V=800.0 PL=0
MOVL C00647 V=800.0 PL=0
MOVL C00648 V=800.0 PL=0
MOVL C00649 V=800.0 PL=0
MOVL C00650 V=800.0 PL=0
MOVL C00651 V=800.0 PL=0
MOVL C00652 V=800.0 PL=0
MOVL C00653 V=800.0 PL=0
MOVL C00654 V=800.0 PL=0
MOVL C00655 V=800.0 PL=0
MOVL C00656 V=800.0 PL=0
MOVL C00657 V=800.0 PL=0
MOVL C00658 V=800.0 PL=0
MOVL C00659 V=800.0 PL=0
MOVL C00660 V=800.0 PL=0
MOVL C00661 V=800.0 PL=0
MOVL C00662 V=800.0 PL=0
MOVL C00663 V=800.0 PL=0
MOVL C00664 V=800.0 PL=0
MOVL C00665 V=800.0 PL=0
MOVL C00666 V=800.0 PL=0
MOVL C00667 V=800.0 PL=0
MOVL C00668 V=800.0 PL=0
MOVL C00669 V=800.0 PL=0
MOVL C00670 V=800.0 PL=0
MOVL C00671 V=800.0 PL=0
MOVL C00672 V=800.0 PL=0
MOVL C00673 V=800.0 PL=0
MOVL C00674 V=800.0 PL=0
MOVL C00675 V=800.0 PL=0
MOVL C00676 V=800.0 PL=0
MOVL C00677 V=800.0 PL=0
MOVL C00678 V=800.0 PL=0
MOVL C00679 V=800.0 PL=0
MOVL C00680 V=800.0 PL=0
MOVL C00681 V=800.0 PL=0
MOVL C00682 V=800.0 PL=0
MOVL C00683 V=800.0 PL=0
MOVL C00684 V=800.0 PL=0
MOVL C00685 V=800.0 PL=0
MOVL C00686 V=800.0 PL=0
MOVL C00687 V=800.0 PL=0
MOVL C00688 V=800.0 PL=0
MOVL C00689 V=800.0 PL=0
MOVL C00690 V=800.0 PL=0
MOVL C00691 V=800.0 PL=0
MOVL C00692 V=800.0 PL=0
MOVL C00693 V=800.0 PL=0
MOVL C00694 V=800.0 PL=0
MOVL C00695 V=800.0 PL=0
MOVL C00696 V=800.0 PL=0
MOVL C00697 V=800.0 PL=0
MOVL C00698 V=800.0 PL=0
MOVL C00699 V=800.0 PL=0
MOVL C00700 V=800.0 PL=0
MOVL C00701 V=800.0 PL=0
MOVL C00702 V=800.0 PL=0
MOVL C00703 V=800.0 PL=0
MOVL C00704 V=800.0 PL=0
MOVL C00705 V=800.0 PL=0
MOVL C00706 V=800.0 PL=0
MOVL C00707 V=800.0 PL=0
MOVL C00708 V=800.0 PL=0
MOVL C00709 V=800.0 PL=0
MOVL C00710 V=800.0 PL=0
MOVL C00711 V=800.0 PL=0
MOVL C00712 V=800.0 PL=0
MOVL C00713 V=800.0 PL=0
MOVL C00714 V=800.0 PL=0
MOVL C00715 V=800.0 PL=0
MOVL C00716 V=800.0 PL=0
MOVL C00717 V=800.0 PL=0
MOVL C00718 V=800.0 PL=0
MOVL C00719 V=800.0 PL=0
MOVL C00720 V=800.0 PL=0
MOVL C00721 V=800.0 PL=0
MOVL C00722 V=800.0 PL=0
MOVL C00723 V=800.0 PL=0
MOVL C00724 V=800.0 PL=0
MOVL C00725 V=800.0 PL=0
MOVL C00726 V=800.0 PL=0
MOVL C00727 V=800.0 PL=0
MOVL C00728 V=800.0 PL=0
MOVL C00729 V=800.0 PL=0
MOVL C00730 V=800.0 PL=0
MOVL C00731 V=800.0 PL=0
MOVL C00732 V=800.0 PL=0
MOVL C00733 V=800.0 PL=0
MOVL C00734 V=800.0 PL=0
MOVL C00735 V=800.0 PL=0
MOVL C00736 V=800.0 PL=0
MOVL C00737 V=800.0 PL=0
MOVL C00738 V=800.0 PL=0
MOVL C00739 V=800.0 PL=0
MOVL C00740 V=800.0 PL=0
MOVL C00741 V=800.0 PL=0
MOVL C00742 V=800.0 PL=0
MOVL C00743 V=800.0 PL=0
MOVL C00744 V=800.0 PL=0
MOVL C00745 V=800.0 PL=0
MOVL C00746 V=800.0 PL=0
MOVL C00747 V=800.0 PL=0
MOVL C00748 V=800.0 PL=0
MOVL C00749 V=800.0 PL=0
MOVL C00750 V=800.0 PL=0
MOVL C00751 V=800.0 PL=0
MOVL C00752 V=800.0 PL=0
MOVL C00753 V=800.0 PL=0
MOVL C00754 V=800.0 PL=0
MOVL C00755 V=800.0 PL=0
MOVL C00756 V=800.0 PL=0
MOVL C00757 V=800.0 PL=0
MOVL C00758 V=800.0 PL=0
MOVL C00759 V=800.0 PL=0
MOVL C00760 V=800.0 PL=0
MOVL C00761 V=800.0 PL=0
MOVL C00762 V=800.0 PL=0
MOVL C00763 V=800.0 PL=0
MOVL C00764 V=800.0 PL=0
MOVL C00765 V=800.0 PL=0
MOVL C00766 V=800.0 PL=0
MOVL C00767 V=800.0 PL=0
MOVL C00768 V=800.0 PL=0
MOVL C00769 V=800.0 PL=0
MOVL C00770 V=800.0 PL=0
MOVL C00771 V=800.0 PL=0
MOVL C00772 V=800.0 PL=0
MOVL C00773 V=800.0 PL=0
MOVL C00774 V=800.0 PL=0
MOVL C00775 V=800.0 PL=0
MOVL C00776 V=800.0 PL=0
MOVL C00777 V=800.0 PL=0
MOVL C00778 V=800.0 PL=0
MOVL C00779 V=800.0 PL=0
MOVL C00780 V=800.0 PL=0
MOVL C00781 V=800.0 PL=0
MOVL C00782 V=800.0 PL=0
MOVL C00783 V=800.0 PL=0
MOVL C00784 V=800.0 PL=0
MOVL C00785 V=800.0 PL=0
MOVL C00786 V=800.0 PL=0
MOVL C00787 V=800.0 PL=0
MOVL C00788 V=800.0 PL=0
MOVL C00789 V=800.0 PL=0
MOVL C00790 V=800.0 PL=0
MOVL C00791 V=800.0 PL=0
MOVL C00792 V=800.0 PL=0
MOVL C00793 V=800.0 PL=0
MOVL C00794 V=800.0 PL=0
MOVL C00795 V=800.0 PL=0
MOVL C00796 V=800.0 PL=0
MOVL C00797 V=800.0 PL=0
MOVL C00798 V=800.0 PL=0
MOVL C00799 V=800.0 PL=0
MOVL C00800 V=800.0 PL=0
MOVL C00801 V=800.0 PL=0
MOVL C00802 V=800.0 PL=0
MOVL C00803 V=800.0 PL=0
MOVL C00804 V=800.0 PL=0
MOVL C00805 V=800.0 PL=0
MOVL C00806 V=800.0 PL=0
MOVL C00807 V=800.0 PL=0
MOVL C00808 V=800.0 PL=0
MOVL C00809 V=800.0 PL=0
MOVL C00810 V=800.0 PL=0
MOVL C00811 V=800.0 PL=0
MOVL C00812 V=800.0 PL=0
MOVL C00813 V=800.0 PL=0
MOVL C00814 V=800.0 PL=0
MOVL C00815 V=800.0 PL=0
MOVL C00816 V=800.0 PL=0
MOVL C00817 V=800.0 PL=0
MOVL C00818 V=800.0 PL=0
MOVL C00819 V=800.0 PL=0
MOVL C00820 V=800.0 PL=0
MOVL C00821 V=800.0 PL=0
MOVL C00822 V=800.0 PL=0
MOVL C00823 V=800.0 PL=0
MOVL C00824 V=800.0 PL=0
MOVL C00825 V=800.0 PL=0
MOVL C00826 V=800.0 PL=0
MOVL C00827 V=800.0 PL=0
MOVL C00828 V=800.0 PL=0
MOVL C00829 V=800.0 PL=0
MOVL C00830 V=800.0 PL=0
MOVL C00831 V=800.0 PL=0
MOVL C00832 V=800.0 PL=0
MOVL C00833 V=800.0 PL=0
MOVL C00834 V=800.0 PL=0
MOVL C00835 V=800.0 PL=0
MOVL C00836 V=800.0 PL=0
MOVL C00837 V=800.0 PL=0
MOVL C00838 V=800.0 PL=0
MOVL C00839 V=800.0 PL=0
MOVL C00840 V=800.0 PL=0
MOVL C00841 V=800.0 PL=0
MOVL C00842 V=800.0 PL=0
MOVL C00843 V=800.0 PL=0
MOVL C00844 V=800.0 PL=0
MOVL C00845 V=800.0 PL=0
MOVL C00846 V=800.0 PL=0
MOVL C00847 V=800.0 PL=0
MOVL C00848 V=800.0 PL=0
MOVL C00849 V=800.0 PL=0
MOVL C00850 V=800.0 PL=0
MOVL C00851 V=800.0 PL=0
MOVL C00852 V=800.0 PL=0
MOVL C00853 V=800.0 PL=0
MOVL C00854 V=800.0 PL=0
MOVL C00855 V=800.0 PL=0
MOVL C00856 V=800.0 PL=0
MOVL C00857 V=800.0 PL=0
MOVL C00858 V=800.0 PL=0
MOVL C00859 V=800.0 PL=0
MOVL C00860 V=800.0 PL=0
MOVL C00861 V=800.0 PL=0
MOVL C00862 V=800.0 PL=0
MOVL C00863 V=800.0 PL=0
MOVL C00864 V=800.0 PL=0
MOVL C00865 V=800.0 PL=0
MOVL C00866 V=800.0 PL=0
MOVL C00867 V=800.0 PL=0
MOVL C00868 V=800.0 PL=0
MOVL C00869 V=800.0 PL=0
MOVL C00870 V=800.0 PL=0
MOVL C00871 V=800.0 PL=0
MOVL C00872 V=800.0 PL=0
MOVL C00873 V=800.0 PL=0
MOVL C00874 V=800.0 PL=0
MOVL C00875 V=800.0 PL=0
MOVL C00876 V=800.0 PL=0
MOVL C00877 V=800.0 PL=0
MOVL C00878 V=800.0 PL=0
MOVL C00879 V=800.0 PL=0
MOVL C00880 V=800.0 PL=0
MOVL C00881 V=800.0 PL=0
MOVL C00882 V=800.0 PL=0
MOVL C00883 V=800.0 PL=0
MOVL C00884 V=800.0 PL=0
MOVL C00885 V=800.0 PL=0
MOVL C00886 V=800.0 PL=0
MOVL C00887 V=800.0 PL=0
MOVL C00888 V=800.0 PL=0
MOVL C00889 V=800.0 PL=0
MOVL C00890 V=800.0 PL=0
MOVL C00891 V=800.0 PL=0
MOVL C00892 V=800.0 PL=0
MOVL C00893 V=800.0 PL=0
MOVL C00894 V=800.0 PL=0
MOVL C00895 V=800.0 PL=0
MOVL C00896 V=800.0 PL=0
MOVL C00897 V=800.0 PL=0
MOVL C00898 V=800.0 PL=0
MOVL C00899 V=800.0 PL=0
MOVL C00900 V=800.0 PL=0
MOVL C00901 V=800.0 PL=0
MOVL C00902 V=800.0 PL=0
MOVL C00903 V=800.0 PL=0
MOVL C00904 V=800.0 PL=0
MOVL C00905 V=800.0 PL=0
MOVL C00906 V=800.0 PL=0
MOVL C00907 V=800.0 PL=0
MOVL C00908 V=800.0 PL=0
MOVL C00909 V=800.0 PL=0
MOVL C00910 V=800.0 PL=0
MOVL C00911 V=800.0 PL=0
MOVL C00912 V=800.0 PL=0
MOVL C00913 V=800.0 PL=0
MOVL C00914 V=800.0 PL=0
MOVL C00915 V=800.0 PL=0
MOVL C00916 V=800.0 PL=0
MOVL C00917 V=800.0 PL=0
MOVL C00918 V=800.0 PL=0
MOVL C00919 V=800.0 PL=0
MOVL C00920 V=800.0 PL=0
MOVL C00921 V=800.0 PL=0
MOVL C00922 V=800.0 PL=0
MOVL C00923 V=800.0 PL=0
MOVL C00924 V=800.0 PL=0
MOVL C00925 V=800.0 PL=0
MOVL C00926 V=800.0 PL=0
MOVL C00927 V=800.0 PL=0
MOVL C00928 V=800.0 PL=0
MOVL C00929 V=800.0 PL=0
MOVL C00930 V=800.0 PL=0
MOVL C00931 V=800.0 PL=0
MOVL C00932 V=800.0 PL=0
MOVL C00933 V=800.0 PL=0
MOVL C00934 V=800.0 PL=0
MOVL C00935 V=800.0 PL=0
MOVL C00936 V=800.0 PL=0
MOVL C00937 V=800.0 PL=0
MOVL C00938 V=800.0 PL=0
MOVL C00939 V=800.0 PL=0
MOVL C00940 V=800.0 PL=0
MOVL C00941 V=800.0 PL=0
MOVL C00942 V=800.0 PL=0
MOVL C00943 V=800.0 PL=0
MOVL C00944 V=800.0 PL=0
MOVL C00945 V=800.0 PL=0
MOVL C00946 V=800.0 PL=0
MOVL C00947 V=800.0 PL=0
MOVL C00948 V=800.0 PL=0
MOVL C00949 V=800.0 PL=0
MOVL C00950 V=800.0 PL=0
MOVL C00951 V=800.0 PL=0
MOVL C00952 V=800.0 PL=0
MOVL C00953 V=800.0 PL=0
MOVL C00954 V=800.0 PL=0
MOVL C00955 V=800.0 PL=0
MOVL C00956 V=800.0 PL=0
MOVL C00957 V=800.0 PL=0
MOVL C00958 V=800.0 PL=0
MOVL C00959 V=800.0 PL=0
MOVL C00960 V=800.0 PL=0
MOVL C00961 V=800.0 PL=0
MOVL C00962 V=800.0 PL=0
MOVL C00963 V=800.0 PL=0
MOVL C00964 V=800.0 PL=0
MOVL C00965 V=800.0 PL=0
MOVL C00966 V=800.0 PL=0
MOVL C00967 V=800.0 PL=0
MOVL C00968 V=800.0 PL=0
MOVL C00969 V=800.0 PL=0
MOVL C00970 V=800.0 PL=0
MOVL C00971 V=800.0 PL=0
MOVL C00972 V=800.0 PL=0
MOVL C00973 V=800.0 PL=0
MOVL C00974 V=800.0 PL=0
MOVL C00975 V=800.0 PL=0
MOVL C00976 V=800.0 PL=0
MOVL C00977 V=800.0 PL=0
MOVL C00978 V=800.0 PL=0
MOVL C00979 V=800.0 PL=0
MOVL C00980 V=800.0 PL=0
MOVL C00981 V=800.0 PL=0
MOVL C00982 V=800.0 PL=0
MOVL C00983 V=800.0 PL=0
MOVL C00984 V=800.0 PL=0
MOVL C00985 V=800.0 PL=0
MOVL C00986 V=800.0 PL=0
MOVL C00987 V=800.0 PL=0
MOVL C00988 V=800.0 PL=0
MOVL C00989 V=800.0 PL=0
MOVL C00990 V=800.0 PL=0
MOVL C00991 V=800.0 PL=0
MOVL C00992 V=800.0 PL=0
MOVL C00993 V=800.0 PL=0
MOVL C00994 V=800.0 PL=0
MOVL C00995 V=800.0 PL=0
MOVL C00996 V=800.0 PL=0
MOVL C00997 V=800.0 PL=0
MOVL C00998 V=800.0 PL=0
MOVL C00999 V=800.0 PL=0
MOVL C01000 V=800.0 PL=0
MOVL C01001 V=800.0 PL=0
MOVL C01002 V=800.0 PL=0
MOVL C01003 V=800.0 PL=0
MOVL C01004 V=800.0 PL=0
MOVL C01005 V=800.0 PL=0
MOVL C01006 V=800.0 PL=0
MOVL C01007 V=800.0 PL=0
MOVL C01008 V=800.0 PL=0
MOVL C01009 V=800.0 PL=0
MOVL C01010 V=800.0 PL=0
MOVL C01011 V=800.0 PL=0
MOVL C01012 V=800.0 PL=0
MOVL C01013 V=800.0 PL=0
MOVL C01014 V=800.0 PL=0
MOVL C01015 V=800.0 PL=0
MOVL C01016 V=800.0 PL=0
MOVL C01017 V=800.0 PL=0
MOVL C01018 V=800.0 PL=0
MOVL C01019 V=800.0 PL=0
MOVL C01020 V=800.0 PL=0
MOVL C01021 V=800.0 PL=0
MOVL C01022 V=800.0 PL=0
MOVL C01023 V=800.0 PL=0
MOVL C01024 V=800.0 PL=0
MOVL C01025 V=800.0 PL=0
MOVL C01026 V=800.0 PL=0
MOVL C01027 V=800.0 PL=0
MOVL C01028 V=800.0 PL=0
MOVL C01029 V=800.0 PL=0
MOVL C01030 V=800.0 PL=0
MOVL C01031 V=800.0 PL=0
MOVL C01032 V=800.0 PL=0
MOVL C01033 V=800.0 PL=0
MOVL C01034 V=800.0 PL=0
MOVL C01035 V=800.0 PL=0
MOVL C01036 V=800.0 PL=0
MOVL C01037 V=800.0 PL=0
MOVL C01038 V=800.0 PL=0
MOVL C01039 V=800.0 PL=0
MOVL C01040 V=800.0 PL=0
MOVL C01041 V=800.0 PL=0
MOVL C01042 V=800.0 PL=0
MOVL C01043 V=800.0 PL=0
MOVL C01044 V=800.0 PL=0
MOVL C01045 V=800.0 PL=0
MOVL C01046 V=800.0 PL=0
MOVL C01047 V=800.0 PL=0
MOVL C01048 V=800.0 PL=0
MOVL C01049 V=800.0 PL=0
MOVL C01050 V=800.0 PL=0
MOVL C01051 V=800.0 PL=0
MOVL C01052 V=800.0 PL=0
MOVL C01053 V=800.0 PL=0
MOVL C01054 V=800.0 PL=0
MOVL C01055 V=800.0 PL=0
MOVL C01056 V=800.0 PL=0
MOVL C01057 V=800.0 PL=0
MOVL C01058 V=800.0 PL=0
MOVL C01059 V=800.0 PL=0
MOVL C01060 V=800.0 PL=0
MOVL C01061 V=800.0 PL=0
MOVL C01062 V=800.0 PL=0
MOVL C01063 V=800.0 PL=0
MOVL C01064 V=800.0 PL=0
MOVL C01065 V=800.0 PL=0
MOVL C01066 V=800.0 PL=0
MOVL C01067 V=800.0 PL=0
MOVL C01068 V=800.0 PL=0
MOVL C01069 V=800.0 PL=0
MOVL C01070 V=800.0 PL=0
MOVL C01071 V=800.0 PL=0
MOVL C01072 V=800.0 PL=0
MOVL C01073 V=800.0 PL=0
MOVL C01074 V=800.0 PL=0
MOVL C01075 V=800.0 PL=0
MOVL C01076 V=800.0 PL=0
MOVL C01077 V=800.0 PL=0
MOVL C01078 V=800.0 PL=0
MOVL C01079 V=800.0 PL=0
MOVL C01080 V=800.0 PL=0
MOVL C01081 V=800.0 PL=0
MOVL C01082 V=800.0 PL=0
MOVL C01083 V=800.0 PL=0
MOVL C01084 V=800.0 PL=0
MOVL C01085 V=800.0 PL=0
MOVL C01086 V=800.0 PL=0
MOVL C01087 V=800.0 PL=0
MOVL C01088 V=800.0 PL=0
MOVL C01089 V=800.0 PL=0
MOVL C01090 V=800.0 PL=0
MOVL C01091 V=800.0 PL=0
MOVL C01092 V=800.0 PL=0
MOVL C01093 V=800.0 PL=0
MOVL C01094 V=800.0 PL=0
MOVL C01095 V=800.0 PL=0
MOVL C01096 V=800.0 PL=0
MOVL C01097 V=800.0 PL=0
MOVL C01098 V=800.0 PL=0
MOVL C01099 V=800.0 PL=0
MOVL C01100 V=800.0 PL=0
MOVL C01101 V=800.0 PL=0
MOVL C01102 V=800.0 PL=0
MOVL C01103 V=800.0 PL=0
MOVL C01104 V=800.0 PL=0
MOVL C01105 V=800.0 PL=0
MOVL C01106 V=800.0 PL=0
MOVL C01107 V=800.0 PL=0
MOVL C01108 V=800.0 PL=0
MOVL C01109 V=800.0 PL=0
MOVL C01110 V=800.0 PL=0
MOVL C01111 V=800.0 PL=0
MOVL C01112 V=800.0 PL=0
MOVL C01113 V=800.0 PL=0
MOVL C01114 V=800.0 PL=0
MOVL C01115 V=800.0 PL=0
MOVL C01116 V=800.0 PL=0
MOVL C01117 V=800.0 PL=0
MOVL C01118 V=800.0 PL=0
MOVL C01119 V=800.0 PL=0
MOVL C01120 V=800.0 PL=0
MOVL C01121 V=800.0 PL=0
MOVL C01122 V=800.0 PL=0
MOVL C01123 V=800.0 PL=0
MOVL C01124 V=800.0 PL=0
MOVL C01125 V=800.0 PL=0
MOVL C01126 V=800.0 PL=0
MOVL C01127 V=800.0 PL=0
MOVL C01128 V=800.0 PL=0
MOVL C01129 V=800.0 PL=0
MOVL C01130 V=800.0 PL=0
MOVL C01131 V=800.0 PL=0
MOVL C01132 V=800.0 PL=0
MOVL C01133 V=800.0 PL=0
MOVL C01134 V=800.0 PL=0
MOVL C01135 V=800.0 PL=0
MOVL C01136 V=800.0 PL=0
MOVL C01137 V=800.0 PL=0
MOVL C01138 V=800.0 PL=0
MOVL C01139 V=800.0 PL=0
MOVL C01140 V=800.0 PL=0
MOVL C01141 V=800.0 PL=0
MOVL C01142 V=800.0 PL=0
MOVL C01143 V=800.0 PL=0
MOVL C01144 V=800.0 PL=0
MOVL C01145 V=800.0 PL=0
MOVL C01146 V=800.0 PL=0
MOVL C01147 V=800.0 PL=0
MOVL C01148 V=800.0 PL=0
MOVL C01149 V=800.0 PL=0
MOVL C01150 V=800.0 PL=0
MOVL C01151 V=800.0 PL=0
MOVL C01152 V=800.0 PL=0
MOVL C01153 V=800.0 PL=0
MOVL C01154 V=800.0 PL=0
MOVL C01155 V=800.0 PL=0
MOVL C01156 V=800.0 PL=0
MOVL C01157 V=800.0 PL=0
MOVL C01158 V=800.0 PL=0
MOVL C01159 V=800.0 PL=0
MOVL C01160 V=800.0 PL=0
MOVL C01161 V=800.0 PL=0
MOVL C01162 V=800.0 PL=0
MOVL C01163 V=800.0 PL=0
MOVL C01164 V=800.0 PL=0
MOVL C01165 V=800.0 PL=0
MOVL C01166 V=800.0 PL=0
MOVL C01167 V=800.0 PL=0
MOVL C01168 V=800.0 PL=0
MOVL C01169 V=800.0 PL=0
MOVL C01170 V=800.0 PL=0
MOVL C01171 V=800.0 PL=0
MOVL C01172 V=800.0 PL=0
MOVL C01173 V=800.0 PL=0
MOVL C01174 V=800.0 PL=0
MOVL C01175 V=800.0 PL=0
MOVL C01176 V=800.0 PL=0
MOVL C01177 V=800.0 PL=0
MOVL C01178 V=800.0 PL=0
MOVL C01179 V=800.0 PL=0
MOVL C01180 V=800.0 PL=0
MOVL C01181 V=800.0 PL=0
MOVL C01182 V=800.0 PL=0
MOVL C01183 V=800.0 PL=0
MOVL C01184 V=800.0 PL=0
MOVL C01185 V=800.0 PL=0
MOVL C01186 V=800.0 PL=0
MOVL C01187 V=800.0 PL=0
MOVL C01188 V=800.0 PL=0
MOVL C01189 V=800.0 PL=0
MOVL C01190 V=800.0 PL=0
MOVL C01191 V=800.0 PL=0
MOVL C01192 V=800.0 PL=0
MOVL C01193 V=800.0 PL=0
MOVL C01194 V=800.0 PL=0
MOVL C01195 V=800.0 PL=0
MOVL C01196 V=800.0 PL=0
MOVL C01197 V=800.0 PL=0
MOVL C01198 V=800.0 PL=0
MOVL C01199 V=800.0 PL=0
MOVL C01200 V=800.0 PL=0
MOVL C01201 V=800.0 PL=0
MOVL C01202 V=800.0 PL=0
MOVL C01203 V=800.0 PL=0
MOVL C01204 V=800.0 PL=0
MOVL C01205 V=800.0 PL=0
MOVL C01206 V=800.0 PL=0
MOVL C01207 V=800.0 PL=0
MOVL C01208 V=800.0 PL=0
MOVL C01209 V=800.0 PL=0
MOVL C01210 V=800.0 PL=0
MOVL C01211 V=800.0 PL=0
MOVL C01212 V=800.0 PL=0
MOVL C01213 V=800.0 PL=0
MOVL C01214 V=800.0 PL=0
MOVL C01215 V=800.0 PL=0
MOVL C01216 V=800.0 PL=0
MOVL C01217 V=800.0 PL=0
MOVL C01218 V=800.0 PL=0
MOVL C01219 V=800.0 PL=0
MOVL C01220 V=800.0 PL=0
MOVL C01221 V=800.0 PL=0
MOVL C01222 V=800.0 PL=0
MOVL C01223 V=800.0 PL=0
MOVL C01224 V=800.0 PL=0
MOVL C01225 V=800.0 PL=0
MOVL C01226 V=800.0 PL=0
MOVL C01227 V=800.0 PL=0
MOVL C01228 V=800.0 PL=0
MOVL C01229 V=800.0 PL=0
MOVL C01230 V=800.0 PL=0
MOVL C01231 V=800.0 PL=0
MOVL C01232 V=800.0 PL=0
MOVL C01233 V=800.0 PL=0
MOVL C01234 V=800.0 PL=0
MOVL C01235 V=800.0 PL=0
MOVL C01236 V=800.0 PL=0
MOVL C01237 V=800.0 PL=0
MOVL C01238 V=800.0 PL=0
MOVL C01239 V=800.0 PL=0
MOVL C01240 V=800.0 PL=0
MOVL C01241 V=800.0 PL=0
MOVL C01242 V=800.0 PL=0
MOVL C01243 V=800.0 PL=0
MOVL C01244 V=800.0 PL=0
MOVL C01245 V=800.0 PL=0
MOVL C01246 V=800.0 PL=0
MOVL C01247 V=800.0 PL=0
MOVL C01248 V=800.0 PL=0
MOVL C01249 V=800.0 PL=0
MOVL C01250 V=800.0 PL=0
MOVL C01251 V=800.0 PL=0
MOVL C01252 V=800.0 PL=0
MOVL C01253 V=800.0 PL=0
MOVL C01254 V=800.0 PL=0
MOVL C01255 V=800.0 PL=0
MOVL C01256 V=800.0 PL=0
MOVL C01257 V=800.0 PL=0
MOVL C01258 V=800.0 PL=0
MOVL C01259 V=800.0 PL=0
MOVL C01260 V=800.0 PL=0
MOVL C01261 V=800.0 PL=0
MOVL C01262 V=800.0 PL=0
MOVL C01263 V=800.0 PL=0
MOVL C01264 V=800.0 PL=0
MOVL C01265 V=800.0 PL=0
MOVL C01266 V=800.0 PL=0
MOVL C01267 V=800.0 PL=0
MOVL C01268 V=800.0 PL=0
MOVL C01269 V=800.0 PL=0
MOVL C01270 V=800.0 PL=0
MOVL C01271 V=800.0 PL=0
MOVL C01272 V=800.0 PL=0
MOVL C01273 V=800.0 PL=0
MOVL C01274 V=800.0 PL=0
MOVL C01275 V=800.0 PL=0
MOVL C01276 V=800.0 PL=0
MOVL C01277 V=800.0 PL=0
MOVL C01278 V=800.0 PL=0
MOVL C01279 V=800.0 PL=0
MOVL C01280 V=800.0 PL=0
MOVL C01281 V=800.0 PL=0
MOVL C01282 V=800.0 PL=0
MOVL C01283 V=800.0 PL=0
MOVL C01284 V=800.0 PL=0
MOVL C01285 V=800.0 PL=0
MOVL C01286 V=800.0 PL=0
MOVL C01287 V=800.0 PL=0
MOVL C01288 V=800.0 PL=0
MOVL C01289 V=800.0 PL=0
MOVL C01290 V=800.0 PL=0
MOVL C01291 V=800.0 PL=0
MOVL C01292 V=800.0 PL=0
MOVL C01293 V=800.0 PL=0
MOVL C01294 V=800.0 PL=0
MOVL C01295 V=800.0 PL=0
MOVL C01296 V=800.0 PL=0
MOVL C01297 V=800.0 PL=0
MOVL C01298 V=800.0 PL=0
MOVL C01299 V=800.0 PL=0
MOVL C01300 V=800.0 PL=0
MOVL C01301 V=800.0 PL=0
MOVL C01302 V=800.0 PL=0
MOVL C01303 V=800.0 PL=0
MOVL C01304 V=800.0 PL=0
MOVL C01305 V=800.0 PL=0
MOVL C01306 V=800.0 PL=0
MOVL C01307 V=800.0 PL=0
MOVL C01308 V=800.0 PL=0
MOVL C01309 V=800.0 PL=0
MOVL C01310 V=800.0 PL=0
MOVL C01311 V=800.0 PL=0
MOVL C01312 V=800.0 PL=0
MOVL C01313 V=800.0 PL=0
MOVL C01314 V=800.0 PL=0
MOVL C01315 V=800.0 PL=0
MOVL C01316 V=800.0 PL=0
MOVL C01317 V=800.0 PL=0
MOVL C01318 V=800.0 PL=0
MOVL C01319 V=800.0 PL=0
MOVL C01320 V=800.0 PL=0
MOVL C01321 V=800.0 PL=0
MOVL C01322 V=800.0 PL=0
MOVL C01323 V=800.0 PL=0
MOVL C01324 V=800.0 PL=0
MOVL C01325 V=800.0 PL=0
MOVL C01326 V=800.0 PL=0
MOVL C01327 V=800.0 PL=0
MOVL C01328 V=800.0 PL=0
MOVL C01329 V=800.0 PL=0
MOVL C01330 V=800.0 PL=0
MOVL C01331 V=800.0 PL=0
MOVL C01332 V=800.0 PL=0
MOVL C01333 V=800.0 PL=0
MOVL C01334 V=800.0 PL=0
MOVL C01335 V=800.0 PL=0
MOVL C01336 V=800.0 PL=0
MOVL C01337 V=800.0 PL=0
MOVL C01338 V=800.0 PL=0
MOVL C01339 V=800.0 PL=0
MOVL C01340 V=800.0 PL=0
MOVL C01341 V=800.0 PL=0
MOVL C01342 V=800.0 PL=0
MOVL C01343 V=800.0 PL=0
MOVL C01344 V=800.0 PL=0
MOVL C01345 V=800.0 PL=0
MOVL C01346 V=800.0 PL=0
MOVL C01347 V=800.0 PL=0
MOVL C01348 V=800.0 PL=0
MOVL C01349 V=800.0 PL=0
MOVL C01350 V=800.0 PL=0
MOVL C01351 V=800.0 PL=0
MOVL C01352 V=800.0 PL=0
MOVL C01353 V=800.0 PL=0
MOVL C01354 V=800.0 PL=0
MOVL C01355 V=800.0 PL=0
MOVL C01356 V=800.0 PL=0
MOVL C01357 V=800.0 PL=0
MOVL C01358 V=800.0 PL=0
MOVL C01359 V=800.0 PL=0
MOVL C01360 V=800.0 PL=0
MOVL C01361 V=800.0 PL=0
MOVL C01362 V=800.0 PL=0
MOVL C01363 V=800.0 PL=0
MOVL C01364 V=800.0 PL=0
MOVL C01365 V=800.0 PL=0
MOVL C01366 V=800.0 PL=0
MOVL C01367 V=800.0 PL=0
MOVL C01368 V=800.0 PL=0
MOVL C01369 V=800.0 PL=0
MOVL C01370 V=800.0 PL=0
MOVL C01371 V=800.0 PL=0
MOVL C01372 V=800.0 PL=0
MOVL C01373 V=800.0 PL=0
MOVL C01374 V=800.0 PL=0
MOVL C01375 V=800.0 PL=0
MOVL C01376 V=800.0 PL=0
MOVL C01377 V=800.0 PL=0
MOVL C01378 V=800.0 PL=0
MOVL C01379 V=800.0 PL=0
MOVL C01380 V=800.0 PL=0
MOVL C01381 V=800.0 PL=0
MOVL C01382 V=800.0 PL=0
MOVL C01383 V=800.0 PL=0
MOVL C01384 V=800.0 PL=0
MOVL C01385 V=800.0 PL=0
MOVL C01386 V=800.0 PL=0
MOVL C01387 V=800.0 PL=0
MOVL C01388 V=800.0 PL=0
MOVL C01389 V=800.0 PL=0
MOVL C01390 V=800.0 PL=0
MOVL C01391 V=800.0 PL=0
MOVL C01392 V=800.0 PL=0
MOVL C01393 V=800.0 PL=0
MOVL C01394 V=800.0 PL=0
MOVL C01395 V=800.0 PL=0
MOVL C01396 V=800.0 PL=0
MOVL C01397 V=800.0 PL=0
MOVL C01398 V=800.0 PL=0
MOVL C01399 V=800.0 PL=0
MOVL C01400 V=800.0 PL=0
MOVL C01401 V=800.0 PL=0
MOVL C01402 V=800.0 PL=0
MOVL C01403 V=800.0 PL=0
MOVL C01404 V=800.0 PL=0
MOVL C01405 V=800.0 PL=0
MOVL C01406 V=800.0 PL=0
MOVL C01407 V=800.0 PL=0
MOVL C01408 V=800.0 PL=0
MOVL C01409 V=800.0 PL=0
MOVL C01410 V=800.0 PL=0
MOVL C01411 V=800.0 PL=0
MOVL C01412 V=800.0 PL=0
MOVL C01413 V=800.0 PL=0
MOVL C01414 V=800.0 PL=0
MOVL C01415 V=800.0 PL=0
MOVL C01416 V=800.0 PL=0
MOVL C01417 V=800.0 PL=0
MOVL C01418 V=800.0 PL=0
MOVL C01419 V=800.0 PL=0
MOVL C01420 V=800.0 PL=0
MOVL C01421 V=800.0 PL=0
MOVL C01422 V=800.0 PL=0
MOVL C01423 V=800.0 PL=0
MOVL C01424 V=800.0 PL=0
MOVL C01425 V=800.0 PL=0
MOVL C01426 V=800.0 PL=0
MOVL C01427 V=800.0 PL=0
MOVL C01428 V=800.0 PL=0
MOVL C01429 V=800.0 PL=0
MOVL C01430 V=800.0 PL=0
MOVL C01431 V=800.0 PL=0
MOVL C01432 V=800.0 PL=0
MOVL C01433 V=800.0 PL=0
MOVL C01434 V=800.0 PL=0
MOVL C01435 V=800.0 PL=0
MOVL C01436 V=800.0 PL=0
MOVL C01437 V=800.0 PL=0
MOVL C01438 V=800.0 PL=0
MOVL C01439 V=800.0 PL=0
MOVL C01440 V=800.0 PL=0
MOVL C01441 V=800.0 PL=0
MOVL C01442 V=800.0 PL=0
MOVL C01443 V=800.0 PL=0
MOVL C01444 V=800.0 PL=0
MOVL C01445 V=800.0 PL=0
MOVL C01446 V=800.0 PL=0
MOVL C01447 V=800.0 PL=0
MOVL C01448 V=800.0 PL=0
MOVL C01449 V=800.0 PL=0
MOVL C01450 V=800.0 PL=0
MOVL C01451 V=800.0 PL=0
MOVL C01452 V=800.0 PL=0
MOVL C01453 V=800.0 PL=0
MOVL C01454 V=800.0 PL=0
MOVL C01455 V=800.0 PL=0
MOVL C01456 V=800.0 PL=0
MOVL C01457 V=800.0 PL=0
MOVL C01458 V=800.0 PL=0
MOVL C01459 V=800.0 PL=0
MOVL C01460 V=800.0 PL=0
MOVL C01461 V=800.0 PL=0
MOVL C01462 V=800.0 PL=0
MOVL C01463 V=800.0 PL=0
MOVL C01464 V=800.0 PL=0
MOVL C01465 V=800.0 PL=0
MOVL C01466 V=800.0 PL=0
MOVL C01467 V=800.0 PL=0
MOVL C01468 V=800.0 PL=0
MOVL C01469 V=800.0 PL=0
MOVL C01470 V=800.0 PL=0
MOVL C01471 V=800.0 PL=0
MOVL C01472 V=800.0 PL=0
MOVL C01473 V=800.0 PL=0
MOVL C01474 V=800.0 PL=0
MOVL C01475 V=800.0 PL=0
MOVL C01476 V=800.0 PL=0
MOVL C01477 V=800.0 PL=0
MOVL C01478 V=800.0 PL=0
MOVL C01479 V=800.0 PL=0
MOVL C01480 V=800.0 PL=0
MOVL C01481 V=800.0 PL=0
MOVL C01482 V=800.0 PL=0
MOVL C01483 V=800.0 PL=0
MOVL C01484 V=800.0 PL=0
MOVL C01485 V=800.0 PL=0
MOVL C01486 V=800.0 PL=0
MOVL C01487 V=800.0 PL=0
MOVL C01488 V=800.0 PL=0
MOVL C01489 V=800.0 PL=0
MOVL C01490 V=800.0 PL=0
MOVL C01491 V=800.0 PL=0
MOVL C01492 V=800.0 PL=0
MOVL C01493 V=800.0 PL=0
MOVL C01494 V=800.0 PL=0
MOVL C01495 V=800.0 PL=0
MOVL C01496 V=800.0 PL=0
MOVL C01497 V=800.0 PL=0
MOVL C01498 V=800.0 PL=0
MOVL C01499 V=800.0 PL=0
MOVL C01500 V=800.0 PL=0
MOVL C01501 V=800.0 PL=0
MOVL C01502 V=800.0 PL=0
MOVL C01503 V=800.0 PL=0
MOVL C01504 V=800.0 PL=0
MOVL C01505 V=800.0 PL=0
MOVL C01506 V=800.0 PL=0
MOVL C01507 V=800.0 PL=0
MOVL C01508 V=800.0 PL=0
MOVL C01509 V=800.0 PL=0
MOVL C01510 V=800.0 PL=0
MOVL C01511 V=800.0 PL=0
MOVL C01512 V=800.0 PL=0
MOVL C01513 V=800.0 PL=0
MOVL C01514 V=800.0 PL=0
MOVL C01515 V=800.0 PL=0
MOVL C01516 V=800.0 PL=0
MOVL C01517 V=800.0 PL=0
MOVL C01518 V=800.0 PL=0
MOVL C01519 V=800.0 PL=0
MOVL C01520 V=800.0 PL=0
MOVL C01521 V=800.0 PL=0
MOVL C01522 V=800.0 PL=0
MOVL C01523 V=800.0 PL=0
MOVL C01524 V=800.0 PL=0
MOVL C01525 V=800.0 PL=0
MOVL C01526 V=800.0 PL=0
MOVL C01527 V=800.0 PL=0
MOVL C01528 V=800.0 PL=0
MOVL C01529 V=800.0 PL=0
MOVL C01530 V=800.0 PL=0
MOVL C01531 V=800.0 PL=0
MOVL C01532 V=800.0 PL=0
MOVL C01533 V=800.0 PL=0
MOVL C01534 V=800.0 PL=0
MOVL C01535 V=800.0 PL=0
MOVL C01536 V=800.0 PL=0
MOVL C01537 V=800.0 PL=0
MOVL C01538 V=800.0 PL=0
MOVL C01539 V=800.0 PL=0
MOVL C01540 V=800.0 PL=0
MOVL C01541 V=800.0 PL=0
MOVL C01542 V=800.0 PL=0
MOVL C01543 V=800.0 PL=0
MOVL C01544 V=800.0 PL=0
MOVL C01545 V=800.0 PL=0
MOVL C01546 V=800.0 PL=0
MOVL C01547 V=800.0 PL=0
MOVL C01548 V=800.0 PL=0
MOVL C01549 V=800.0 PL=0
MOVL C01550 V=800.0 PL=0
MOVL C01551 V=800.0 PL=0
MOVL C01552 V=800.0 PL=0
MOVL C01553 V=800.0 PL=0
MOVL C01554 V=800.0 PL=0
MOVL C01555 V=800.0 PL=0
MOVL C01556 V=800.0 PL=0
MOVL C01557 V=800.0 PL=0
MOVL C01558 V=800.0 PL=0
MOVL C01559 V=800.0 PL=0
MOVL C01560 V=800.0 PL=0
MOVL C01561 V=800.0 PL=0
MOVL C01562 V=800.0 PL=0
MOVL C01563 V=800.0 PL=0
MOVL C01564 V=800.0 PL=0
MOVL C01565 V=800.0 PL=0
MOVL C01566 V=800.0 PL=0
MOVL C01567 V=800.0 PL=0
MOVL C01568 V=800.0 PL=0
MOVL C01569 V=800.0 PL=0
MOVL C01570 V=800.0 PL=0
MOVL C01571 V=800.0 PL=0
MOVL C01572 V=800.0 PL=0
MOVL C01573 V=800.0 PL=0
MOVL C01574 V=800.0 PL=0
MOVL C01575 V=800.0 PL=0
MOVL C01576 V=800.0 PL=0
MOVL C01577 V=800.0 PL=0
MOVL C01578 V=800.0 PL=0
MOVL C01579 V=800.0 PL=0
MOVL C01580 V=800.0 PL=0
MOVL C01581 V=800.0 PL=0
MOVL C01582 V=800.0 PL=0
MOVL C01583 V=800.0 PL=0
MOVL C01584 V=800.0 PL=0
MOVL C01585 V=800.0 PL=0
MOVL C01586 V=800.0 PL=0
MOVL C01587 V=800.0 PL=0
MOVL C01588 V=800.0 PL=0
MOVL C01589 V=800.0 PL=0
MOVL C01590 V=800.0 PL=0
MOVL C01591 V=800.0 PL=0
MOVL C01592 V=800.0 PL=0
MOVL C01593 V=800.0 PL=0
MOVL C01594 V=800.0 PL=0
MOVL C01595 V=800.0 PL=0
MOVL C01596 V=800.0 PL=0
MOVL C01597 V=800.0 PL=0
MOVL C01598 V=800.0 PL=0
MOVL C01599 V=800.0 PL=0
MOVL C01600 V=800.0 PL=0
MOVL C01601 V=800.0 PL=0
MOVL C01602 V=800.0 PL=0
MOVL C01603 V=800.0 PL=0
MOVL C01604 V=800.0 PL=0
MOVL C01605 V=800.0 PL=0
MOVL C01606 V=800.0 PL=0
MOVL C01607 V=800.0 PL=0
MOVL C01608 V=800.0 PL=0
MOVL C01609 V=800.0 PL=0
MOVL C01610 V=800.0 PL=0
MOVL C01611 V=800.0 PL=0
MOVL C01612 V=800.0 PL=0
MOVL C01613 V=800.0 PL=0
MOVL C01614 V=800.0 PL=0
MOVL C01615 V=800.0 PL=0
MOVL C01616 V=800.0 PL=0
MOVL C01617 V=800.0 PL=0
MOVL C01618 V=800.0 PL=0
MOVL C01619 V=800.0 PL=0
MOVL C01620 V=800.0 PL=0
MOVL C01621 V=800.0 PL=0
MOVL C01622 V=800.0 PL=0
MOVL C01623 V=800.0 PL=0
MOVL C01624 V=800.0 PL=0
MOVL C01625 V=800.0 PL=0
MOVL C01626 V=800.0 PL=0
MOVL C01627 V=800.0 PL=0
MOVL C01628 V=800.0 PL=0
MOVL C01629 V=800.0 PL=0
MOVL C01630 V=800.0 PL=0
MOVL C01631 V=800.0 PL=0
MOVL C01632 V=800.0 PL=0
MOVL C01633 V=800.0 PL=0
MOVL C01634 V=800.0 PL=0
MOVL C01635 V=800.0 PL=0
MOVL C01636 V=800.0 PL=0
MOVL C01637 V=800.0 PL=0
MOVL C01638 V=800.0 PL=0
MOVL C01639 V=800.0 PL=0
MOVL C01640 V=800.0 PL=0
MOVL C01641 V=800.0 PL=0
MOVL C01642 V=800.0 PL=0
MOVL C01643 V=800.0 PL=0
MOVL C01644 V=800.0 PL=0
MOVL C01645 V=800.0 PL=0
MOVL C01646 V=800.0 PL=0
MOVL C01647 V=800.0 PL=0
MOVL C01648 V=800.0 PL=0
MOVL C01649 V=800.0 PL=0
MOVL C01650 V=800.0 PL=0
MOVL C01651 V=800.0 PL=0
MOVL C01652 V=800.0 PL=0
MOVL C01653 V=800.0 PL=0
MOVL C01654 V=800.0 PL=0
MOVL C01655 V=800.0 PL=0
MOVL C01656 V=800.0 PL=0
MOVL C01657 V=800.0 PL=0
MOVL C01658 V=800.0 PL=0
MOVL C01659 V=800.0 PL=0
MOVL C01660 V=800.0 PL=0
MOVL C01661 V=800.0 PL=0
MOVL C01662 V=800.0 PL=0
MOVL C01663 V=800.0 PL=0
MOVL C01664 V=800.0 PL=0
MOVL C01665 V=800.0 PL=0
MOVL C01666 V=800.0 PL=0
MOVL C01667 V=800.0 PL=0
MOVL C01668 V=800.0 PL=0
MOVL C01669 V=800.0 PL=0
MOVL C01670 V=800.0 PL=0
MOVL C01671 V=800.0 PL=0
MOVL C01672 V=800.0 PL=0
MOVL C01673 V=800.0 PL=0
MOVL C01674 V=800.0 PL=0
MOVL C01675 V=800.0 PL=0
MOVL C01676 V=800.0 PL=0
MOVL C01677 V=800.0 PL=0
MOVL C01678 V=800.0 PL=0
MOVL C01679 V=800.0 PL=0
MOVL C01680 V=800.0 PL=0
MOVL C01681 V=800.0 PL=0
MOVL C01682 V=800.0 PL=0
MOVL C01683 V=800.0 PL=0
MOVL C01684 V=800.0 PL=0
MOVL C01685 V=800.0 PL=0
MOVL C01686 V=800.0 PL=0
MOVL C01687 V=800.0 PL=0
MOVL C01688 V=800.0 PL=0
MOVL C01689 V=800.0 PL=0
MOVL C01690 V=800.0 PL=0
MOVL C01691 V=800.0 PL=0
MOVL C01692 V=800.0 PL=0
MOVL C01693 V=800.0 PL=0
MOVL C01694 V=800.0 PL=0
MOVL C01695 V=800.0 PL=0
MOVL C01696 V=800.0 PL=0
MOVL C01697 V=800.0 PL=0
MOVL C01698 V=800.0 PL=0
MOVL C01699 V=800.0 PL=0
MOVL C01700 V=800.0 PL=0
MOVL C01701 V=800.0 PL=0
MOVL C01702 V=800.0 PL=0
MOVL C01703 V=800.0 PL=0
MOVL C01704 V=800.0 PL=0
MOVL C01705 V=800.0 PL=0
MOVL C01706 V=800.0 PL=0
MOVL C01707 V=800.0 PL=0
MOVL C01708 V=800.0 PL=0
MOVL C01709 V=800.0 PL=0
MOVL C01710 V=800.0 PL=0
MOVL C01711 V=800.0 PL=0
MOVL C01712 V=800.0 PL=0
MOVL C01713 V=800.0 PL=0
MOVL C01714 V=800.0 PL=0
MOVL C01715 V=800.0 PL=0
MOVL C01716 V=800.0 PL=0
MOVL C01717 V=800.0 PL=0
MOVL C01718 V=800.0 PL=0
MOVL C01719 V=800.0 PL=0
MOVL C01720 V=800.0 PL=0
MOVL C01721 V=800.0 PL=0
MOVL C01722 V=800.0 PL=0
MOVL C01723 V=800.0 PL=0
MOVL C01724 V=800.0 PL=0
MOVL C01725 V=800.0 PL=0
MOVL C01726 V=800.0 PL=0
MOVL C01727 V=800.0 PL=0
MOVL C01728 V=800.0 PL=0
MOVL C01729 V=800.0 PL=0
MOVL C01730 V=800.0 PL=0
MOVL C01731 V=800.0 PL=0
MOVL C01732 V=800.0 PL=0
MOVL C01733 V=800.0 PL=0
MOVL C01734 V=800.0 PL=0
MOVL C01735 V=800.0 PL=0
MOVL C01736 V=800.0 PL=0
MOVL C01737 V=800.0 PL=0
MOVL C01738 V=800.0 PL=0
MOVL C01739 V=800.0 PL=0
MOVL C01740 V=800.0 PL=0
MOVL C01741 V=800.0 PL=0
MOVL C01742 V=800.0 PL=0
MOVL C01743 V=800.0 PL=0
MOVL C01744 V=800.0 PL=0
MOVL C01745 V=800.0 PL=0
MOVL C01746 V=800.0 PL=0
MOVL C01747 V=800.0 PL=0
MOVL C01748 V=800.0 PL=0
MOVL C01749 V=800.0 PL=0
MOVL C01750 V=800.0 PL=0
MOVL C01751 V=800.0 PL=0
MOVL C01752 V=800.0 PL=0
MOVL C01753 V=800.0 PL=0
MOVL C01754 V=800.0 PL=0
MOVL C01755 V=800.0 PL=0
MOVL C01756 V=800.0 PL=0
MOVL C01757 V=800.0 PL=0
MOVL C01758 V=800.0 PL=0
MOVL C01759 V=800.0 PL=0
MOVL C01760 V=800.0 PL=0
MOVL C01761 V=800.0 PL=0
MOVL C01762 V=800.0 PL=0
MOVL C01763 V=800.0 PL=0
MOVL C01764 V=800.0 PL=0
MOVL C01765 V=800.0 PL=0
MOVL C01766 V=800.0 PL=0
MOVL C01767 V=800.0 PL=0
MOVL C01768 V=800.0 PL=0
MOVL C01769 V=800.0 PL=0
MOVL C01770 V=800.0 PL=0
MOVL C01771 V=800.0 PL=0
MOVL C01772 V=800.0 PL=0
MOVL C01773 V=800.0 PL=0
MOVL C01774 V=800.0 PL=0
MOVL C01775 V=800.0 PL=0
MOVL C01776 V=800.0 PL=0
MOVL C01777 V=800.0 PL=0
MOVL C01778 V=800.0 PL=0
MOVL C01779 V=800.0 PL=0
MOVL C01780 V=800.0 PL=0
MOVL C01781 V=800.0 PL=0
MOVL C01782 V=800.0 PL=0
MOVL C01783 V=800.0 PL=0
MOVL C01784 V=800.0 PL=0
MOVL C01785 V=800.0 PL=0
MOVL C01786 V=800.0 PL=0
MOVL C01787 V=800.0 PL=0
MOVL C01788 V=800.0 PL=0
MOVL C01789 V=800.0 PL=0
MOVL C01790 V=800.0 PL=0
MOVL C01791 V=800.0 PL=0
MOVL C01792 V=800.0 PL=0
MOVL C01793 V=800.0 PL=0
MOVL C01794 V=800.0 PL=0
MOVL C01795 V=800.0 PL=0
MOVL C01796 V=800.0 PL=0
MOVL C01797 V=800.0 PL=0
MOVL C01798 V=800.0 PL=0
MOVL C01799 V=800.0 PL=0
MOVL C01800 V=800.0 PL=0
MOVL C01801 V=800.0 PL=0
MOVL C01802 V=800.0 PL=0
MOVL C01803 V=800.0 PL=0
MOVL C01804 V=800.0 PL=0
MOVL C01805 V=800.0 PL=0
MOVL C01806 V=800.0 PL=0
MOVL C01807 V=800.0 PL=0
MOVL C01808 V=800.0 PL=0
MOVL C01809 V=800.0 PL=0
MOVL C01810 V=800.0 PL=0
MOVL C01811 V=800.0 PL=0
MOVL C01812 V=800.0 PL=0
MOVL C01813 V=800.0 PL=0
MOVL C01814 V=800.0 PL=0
MOVL C01815 V=800.0 PL=0
MOVL C01816 V=800.0 PL=0
MOVL C01817 V=800.0 PL=0
MOVL C01818 V=800.0 PL=0
MOVL C01819 V=800.0 PL=0
MOVL C01820 V=800.0 PL=0
MOVL C01821 V=800.0 PL=0
MOVL C01822 V=800.0 PL=0
MOVL C01823 V=800.0 PL=0
MOVL C01824 V=800.0 PL=0
MOVL C01825 V=800.0 PL=0
MOVL C01826 V=800.0 PL=0
MOVL C01827 V=800.0 PL=0
MOVL C01828 V=800.0 PL=0
MOVL C01829 V=800.0 PL=0
MOVL C01830 V=800.0 PL=0
MOVL C01831 V=800.0 PL=0
MOVL C01832 V=800.0 PL=0
MOVL C01833 V=800.0 PL=0
MOVL C01834 V=800.0 PL=0
MOVL C01835 V=800.0 PL=0
MOVL C01836 V=800.0 PL=0
MOVL C01837 V=800.0 PL=0
MOVL C01838 V=800.0 PL=0
MOVL C01839 V=800.0 PL=0
MOVL C01840 V=800.0 PL=0
MOVL C01841 V=800.0 PL=0
MOVL C01842 V=800.0 PL=0
MOVL C01843 V=800.0 PL=0
MOVL C01844 V=800.0 PL=0
MOVL C01845 V=800.0 PL=0
MOVL C01846 V=800.0 PL=0
MOVL C01847 V=800.0 PL=0
MOVL C01848 V=800.0 PL=0
MOVL C01849 V=800.0 PL=0
MOVL C01850 V=800.0 PL=0
MOVL C01851 V=800.0 PL=0
MOVL C01852 V=800.0 PL=0
MOVL C01853 V=800.0 PL=0
MOVL C01854 V=800.0 PL=0
MOVL C01855 V=800.0 PL=0
MOVL C01856 V=800.0 PL=0
MOVL C01857 V=800.0 PL=0
MOVL C01858 V=800.0 PL=0
MOVL C01859 V=800.0 PL=0
MOVL C01860 V=800.0 PL=0
MOVL C01861 V=800.0 PL=0
MOVL C01862 V=800.0 PL=0
MOVL C01863 V=800.0 PL=0
MOVL C01864 V=800.0 PL=0
MOVL C01865 V=800.0 PL=0
MOVL C01866 V=800.0 PL=0
MOVL C01867 V=800.0 PL=0
MOVL C01868 V=800.0 PL=0
MOVL C01869 V=800.0 PL=0
MOVL C01870 V=800.0 PL=0
MOVL C01871 V=800.0 PL=0
MOVL C01872 V=800.0 PL=0
MOVL C01873 V=800.0 PL=0
MOVL C01874 V=800.0 PL=0
MOVL C01875 V=800.0 PL=0
MOVL C01876 V=800.0 PL=0
MOVL C01877 V=800.0 PL=0
MOVL C01878 V=800.0 PL=0
MOVL C01879 V=800.0 PL=0
MOVL C01880 V=800.0 PL=0
MOVL C01881 V=800.0 PL=0
MOVL C01882 V=800.0 PL=0
MOVL C01883 V=800.0 PL=0
MOVL C01884 V=800.0 PL=0
MOVL C01885 V=800.0 PL=0
MOVL C01886 V=800.0 PL=0
MOVL C01887 V=800.0 PL=0
MOVL C01888 V=800.0 PL=0
MOVL C01889 V=800.0 PL=0
MOVL C01890 V=800.0 PL=0
MOVL C01891 V=800.0 PL=0
MOVL C01892 V=800.0 PL=0
MOVL C01893 V=800.0 PL=0
MOVL C01894 V=800.0 PL=0
MOVL C01895 V=800.0 PL=0
MOVL C01896 V=800.0 PL=0
MOVL C01897 V=800.0 PL=0
MOVL C01898 V=800.0 PL=0
MOVL C01899 V=800.0 PL=0
MOVL C01900 V=800.0 PL=0
MOVL C01901 V=800.0 PL=0
MOVL C01902 V=800.0 PL=0
MOVL C01903 V=800.0 PL=0
MOVL C01904 V=800.0 PL=0
MOVL C01905 V=800.0 PL=0
MOVL C01906 V=800.0 PL=0
MOVL C01907 V=800.0 PL=0
MOVL C01908 V=800.0 PL=0
MOVL C01909 V=800.0 PL=0
MOVL C01910 V=800.0 PL=0
MOVL C01911 V=800.0 PL=0
MOVL C01912 V=800.0 PL=0
MOVL C01913 V=800.0 PL=0
MOVL C01914 V=800.0 PL=0
MOVL C01915 V=800.0 PL=0
MOVL C01916 V=800.0 PL=0
MOVL C01917 V=800.0 PL=0
MOVL C01918 V=800.0 PL=0
MOVL C01919 V=800.0 PL=0
MOVL C01920 V=800.0 PL=0
MOVL C01921 V=800.0 PL=0
MOVL C01922 V=800.0 PL=0
MOVL C01923 V=800.0 PL=0
MOVL C01924 V=800.0 PL=0
MOVL C01925 V=800.0 PL=0
MOVL C01926 V=800.0 PL=0
MOVL C01927 V=800.0 PL=0
MOVL C01928 V=800.0 PL=0
MOVL C01929 V=800.0 PL=0
MOVL C01930 V=800.0 PL=0
MOVL C01931 V=800.0 PL=0
MOVL C01932 V=800.0 PL=0
MOVL C01933 V=800.0 PL=0
MOVL C01934 V=800.0 PL=0
MOVL C01935 V=800.0 PL=0
MOVL C01936 V=800.0 PL=0
MOVL C01937 V=800.0 PL=0
MOVL C01938 V=800.0 PL=0
MOVL C01939 V=800.0 PL=0
MOVL C01940 V=800.0 PL=0
MOVL C01941 V=800.0 PL=0
MOVL C01942 V=800.0 PL=0
MOVL C01943 V=800.0 PL=0
MOVL C01944 V=800.0 PL=0
MOVL C01945 V=800.0 PL=0
MOVL C01946 V=800.0 PL=0
MOVL C01947 V=800.0 PL=0
MOVL C01948 V=800.0 PL=0
MOVL C01949 V=800.0 PL=0
MOVL C01950 V=800.0 PL=0
MOVL C01951 V=800.0 PL=0
MOVL C01952 V=800.0 PL=0
MOVL C01953 V=800.0 PL=0
MOVL C01954 V=800.0 PL=0
MOVL C01955 V=800.0 PL=0
MOVL C01956 V=800.0 PL=0
MOVL C01957 V=800.0 PL=0
MOVL C01958 V=800.0 PL=0
MOVL C01959 V=800.0 PL=0
MOVL C01960 V=800.0 PL=0
MOVL C01961 V=800.0 PL=0
MOVL C01962 V=800.0 PL=0
MOVL C01963 V=800.0 PL=0
MOVL C01964 V=800.0 PL=0
MOVL C01965 V=800.0 PL=0
MOVL C01966 V=800.0 PL=0
MOVL C01967 V=800.0 PL=0
MOVL C01968 V=800.0 PL=0
MOVL C01969 V=800.0 PL=0
MOVL C01970 V=800.0 PL=0
MOVL C01971 V=800.0 PL=0
MOVL C01972 V=800.0 PL=0
MOVL C01973 V=800.0 PL=0
MOVL C01974 V=800.0 PL=0
MOVL C01975 V=800.0 PL=0
MOVL C01976 V=800.0 PL=0
MOVL C01977 V=800.0 PL=0
MOVL C01978 V=800.0 PL=0
MOVL C01979 V=800.0 PL=0
MOVL C01980 V=800.0 PL=0
MOVL C01981 V=800.0 PL=0
MOVL C01982 V=800.0 PL=0
MOVL C01983 V=800.0 PL=0
MOVL C01984 V=800.0 PL=0
MOVL C01985 V=800.0 PL=0
MOVL C01986 V=800.0 PL=0
MOVL C01987 V=800.0 PL=0
MOVL C01988 V=800.0 PL=0
MOVL C01989 V=800.0 PL=0
MOVL C01990 V=800.0 PL=0
MOVL C01991 V=800.0 PL=0
MOVL C01992 V=800.0 PL=0
MOVL C01993 V=800.0 PL=0
MOVL C01994 V=800.0 PL=0
MOVL C01995 V=800.0 PL=0
MOVL C01996 V=800.0 PL=0
MOVL C01997 V=800.0 PL=0
MOVL C01998 V=800.0 PL=0
MOVL C01999 V=800.0 PL=0
MOVL C02000 V=800.0 PL=0
MOVL C02001 V=800.0 PL=0
MOVL C02002 V=800.0 PL=0
MOVL C02003 V=800.0 PL=0
MOVL C02004 V=800.0 PL=0
MOVL C02005 V=800.0 PL=0
MOVL C02006 V=800.0 PL=0
MOVL C02007 V=800.0 PL=0
MOVL C02008 V=800.0 PL=0
MOVL C02009 V=800.0 PL=0
MOVL C02010 V=800.0 PL=0
MOVL C02011 V=800.0 PL=0
MOVL C02012 V=800.0 PL=0
MOVL C02013 V=800.0 PL=0
MOVL C02014 V=800.0 PL=0
MOVL C02015 V=800.0 PL=0
MOVL C02016 V=800.0 PL=0
MOVL C02017 V=800.0 PL=0
MOVL C02018 V=800.0 PL=0
MOVL C02019 V=800.0 PL=0
MOVL C02020 V=800.0 PL=0
MOVL C02021 V=800.0 PL=0
MOVL C02022 V=800.0 PL=0
MOVL C02023 V=800.0 PL=0
MOVL C02024 V=800.0 PL=0
MOVL C02025 V=800.0 PL=0
MOVL C02026 V=800.0 PL=0
MOVL C02027 V=800.0 PL=0
MOVL C02028 V=800.0 PL=0
MOVL C02029 V=800.0 PL=0
MOVL C02030 V=800.0 PL=0
MOVL C02031 V=800.0 PL=0
MOVL C02032 V=800.0 PL=0
MOVL C02033 V=800.0 PL=0
MOVL C02034 V=800.0 PL=0
MOVL C02035 V=800.0 PL=0
MOVL C02036 V=800.0 PL=0
MOVL C02037 V=800.0 PL=0
MOVL C02038 V=800.0 PL=0
MOVL C02039 V=800.0 PL=0
MOVL C02040 V=800.0 PL=0
MOVL C02041 V=800.0 PL=0
